// TwinCAT 3 PLC project tmo_motion
// Title: lcls-plc-tmo-motion
// Company: SLAC
// ProjectVersion: 0.0.0
// ProgramVersion: 3.1.4022.7
// CompilerDefines: K
// libraries:
//   LCLS General, * (SLAC)
//   lcls-twincat-motion, * (SLAC)
//   lcls2-cc-lib, * (SLAC)
//   PMPS, * (SLAC - LCLS)
//   Tc2_MC2, * (Beckhoff Automation GmbH)
//   Tc2_SerialCom, * (Beckhoff Automation GmbH)
//   Tc2_Standard, * (Beckhoff Automation GmbH)
//   Tc2_System, * (Beckhoff Automation GmbH)
//   Tc3_Module, * (Beckhoff Automation GmbH)
// project tree:
//   DUTs/ E_HomeState.TcDUT (not stored)
//   GVLs/ GVL_PMPS.TcGVL (not stored), Main.TcGVL
//   / PlcTask.TcTTO
//   POUs/ PRG_1_PlcTask.TcPOU, PRG_2_PMPS_PRE.TcPOU, PRG_3_PMPS_POST.TcPOU, PRG_4_LOG.TcPOU, PRG_AL1K4_L2SI.TcPOU, PRG_IM2K4_PPM.TcPOU, PRG_IM3K4_PPM.TcPOU, PRG_IM4K4_PPM.TcPOU, PRG_IM5K4_PPM.TcPOU, PRG_LI1K4_IP1.TcPOU, PRG_PF1K4_WFS_TARGET.TcPOU, PRG_SL1K4_SCATTER.TcPOU, PRG_SL2K4_SCATTER.TcPOU, PRG_ST4K4_TMO_TERM.TcPOU, PRG_ST5K4_TMO_TERM_FIXED.TcPOU, PRG_TM1K4.TcPOU (not stored)
//   POUs/temp/ FB_SLITS.TcPOU, FB_SLITS_POWER.TcPOU (not stored), FB_SLITS_SCATTER.TcPOU
// real-time tasks:
//   TASK PlcTask: cycle T#10ms, priority 20, ADS port 350
// motion (NC):
//   TASK NC-Task 1 SAF: cycle T#2ms, priority 4, ADS port 501
//   TASK NC-Task 1 SVB: cycle T#10ms, priority 8, ADS port 511
//   AXIS Axis 1 AL1K4-L2SI-MMS (id 1)
//     Dynamic: AccelerationMaximum=200, DecelerationMaximum=200, Acceleration=200, Deceleration=200, Jerk=500, DelayTime=0.004
//     Velo: Maximum=10
//     TargetPosControl: Range=0.002, Time=2
//     OtherSettings: AllowMotionCmdToSlave=true
//     encoder EncType=29
//       EncPara: ScaleFactorNumerator=5e-05, Offset=-214686.941, MaxCount=#xffffffff, ReferenceSystem=1
//         SoftEndMinControl: Enable=true, Range=-108.74
//         SoftEndMaxControl: Enable=true, Range=-33.49
//         Inc: RefSoftSyncMask=#x0000ffff
//     drive DrvType=24
//       Analog: VeloReferenz=100, ScaleFactorActTorque=0.1
//       TimeComp: TaskDelayCycles=1
//     controller CtrType=2
//       CtrPara: PriorControlFactor=1
//         PosDiffControl: Range=1
//         PID: PosKp=20, PosExtKp=1, PosExtVelo=0.1, DeadBandPosition=0.002
//         Observer: BandWidth=20
//   AXIS Axis 2 (id 2)
//     OtherSettings: AllowMotionCmdToSlave=true
//     encoder EncType=1
//     drive DrvType=5
//       Analog: ScaleFactorActTorque=0.1
//       TimeComp: TaskDelayCycles=1
//     controller CtrType=1
//       CtrPara: PriorControlFactor=1
//         Observer: BandWidth=20
//   AXIS Axis 3 (id 3)
//     OtherSettings: AllowMotionCmdToSlave=true
//     encoder EncType=1
//     drive DrvType=5
//       Analog: ScaleFactorActTorque=0.1
//       TimeComp: TaskDelayCycles=1
//     controller CtrType=1
//       CtrPara: PriorControlFactor=1
//         Observer: BandWidth=20
//   AXIS Axis 4 (id 4)
//     OtherSettings: AllowMotionCmdToSlave=true
//     encoder EncType=1
//     drive DrvType=5
//       Analog: ScaleFactorActTorque=0.1
//       TimeComp: TaskDelayCycles=1
//     controller CtrType=1
//       CtrPara: PriorControlFactor=1
//         Observer: BandWidth=20
//   AXIS Axis 5 (id 5)
//     OtherSettings: AllowMotionCmdToSlave=true
//     encoder EncType=1
//     drive DrvType=5
//       Analog: ScaleFactorActTorque=0.1
//       TimeComp: TaskDelayCycles=1
//     controller CtrType=1
//       CtrPara: PriorControlFactor=1
//         Observer: BandWidth=20
//   AXIS Axis 6 IM1K4-XTES-MMS (id 6)
//     Velo: Maximum=10
//     OtherSettings: AllowMotionCmdToSlave=true
//     encoder EncType=29
//       EncPara: ScaleFactorNumerator=5e-05, Offset=-398.1892, MaxCount=#x00400000, ReferenceSystem=1
//         SoftEndMinControl: Enable=true, Range=-90
//         SoftEndMaxControl: Enable=true
//         Inc: RefSoftSyncMask=#x00000000
//     drive DrvType=24
//       DrvPara: Inverse=true
//         Analog: VeloReferenz=50, ScaleFactorActTorque=0.1
//         TimeComp: TaskDelayCycles=1
//     controller CtrType=2
//       CtrPara: PriorControlFactor=1
//         PosDiffControl: Range=1
//         PID: PosKp=20, PosExtKp=20, DeadBandPosition=0.001
//         Observer: BandWidth=20
//   AXIS Axis 7 IM1K4-XTES-CLZ (id 7)
//     General: UnitName=%
//     Velo: Maximum=10
//     OtherSettings: AllowMotionCmdToSlave=true
//     encoder EncType=4
//       EncPara: ScaleFactorNumerator=0.003, MaxCount=#x0000ffff
//         SoftEndMinControl: Enable=true, Range=-100
//         SoftEndMaxControl: Enable=true, Range=100
//         Inc: RefSoftSyncMask=#x0000ffff
//     drive DrvType=23
//       DrvPara: Inverse=true
//         Analog: VeloReferenz=33, ScaleFactorActTorque=0.1
//         TimeComp: TaskDelayCycles=1
//     controller CtrType=2
//       CtrPara: PriorControlFactor=1
//         PosDiffControl: Range=1
//         PID: PosKp=20, PosExtKp=20, DeadBandPosition=0.1
//         Observer: BandWidth=20
//   AXIS Axis 8 IM1K4-XTES-CLF (id 8)
//     General: UnitName=%
//     Velo: Maximum=10
//     OtherSettings: AllowMotionCmdToSlave=true
//     encoder EncType=4
//       EncPara: ScaleFactorNumerator=0.008, MaxCount=#x0000ffff
//         SoftEndMinControl: Enable=true, Range=-100
//         SoftEndMaxControl: Enable=true, Range=100
//         Inc: RefSoftSyncMask=#x0000ffff
//     drive DrvType=23
//       DrvPara: Inverse=true
//         Analog: VeloReferenz=70, ScaleFactorActTorque=0.1
//         TimeComp: TaskDelayCycles=1
//     controller CtrType=2
//       CtrPara: PriorControlFactor=1
//         PosDiffControl: Range=1
//         PID: PosKp=20, PosExtKp=20, DeadBandPosition=0.1
//         Observer: BandWidth=20
//   AXIS Axis 9 IM2K4-PPM-MMS (id 9)
//     Dynamic: AccelerationMaximum=200, DecelerationMaximum=200, Acceleration=200, Deceleration=200, Jerk=500, DelayTime=0.004
//     Velo: Maximum=65
//     TargetPosControl: Range=0.002, Time=2
//     OtherSettings: AllowMotionCmdToSlave=true
//     encoder EncType=29
//       EncPara: ScaleFactorNumerator=5e-05, Offset=-358.0066, MaxCount=#x00400000, ReferenceSystem=1
//         SoftEndMinControl: Enable=true, Range=-100.57
//         SoftEndMaxControl: Enable=true, Range=-7.67
//         Inc: RefSoftSyncMask=#x00000000
//     drive DrvType=24
//       Analog: VeloReferenz=100, ScaleFactorActTorque=0.1
//       TimeComp: TaskDelayCycles=1
//     controller CtrType=2
//       CtrPara: PriorControlFactor=1
//         PosDiffControl: Range=1
//         PID: PosKp=20, PosExtKp=1, PosExtVelo=0.1, DeadBandPosition=0.002
//         Observer: BandWidth=20
//   AXIS SL1K4-BOTTOM-M10 (id 10)
//     Velo: RefSearch=0.2, RefSync=0.05, Maximum=2.2
//     OtherSettings: AllowMotionCmdToSlave=true
//     encoder EncType=4
//       EncPara: MaxCount=#x0000ffff
//         SoftEndMinControl: Enable=true, Range=-31.51
//         SoftEndMaxControl: Enable=true
//         Inc: RefSoftSyncMask=#x0000ffff
//     drive DrvType=24
//       Analog: VeloReferenz=2, ScaleFactorActTorque=0.1
//       TimeComp: TaskDelayCycles=1
//     controller CtrType=1
//       CtrPara: PriorControlFactor=1
//         PosDiffControl: Range=0.05
//         Observer: BandWidth=20
//   AXIS SL1K4-TOP-M11 (id 11)
//     Velo: RefSearch=0.2, RefSync=0.05, Maximum=2.2
//     OtherSettings: AllowMotionCmdToSlave=true
//     encoder EncType=4
//       EncPara: Inverse=true, MaxCount=#x0000ffff
//         SoftEndMinControl: Enable=true, Range=-31.99
//         SoftEndMaxControl: Enable=true
//         Inc: RefSoftSyncMask=#x0000ffff
//     drive DrvType=24
//       Analog: VeloReferenz=2, ScaleFactorActTorque=0.1
//       TimeComp: TaskDelayCycles=1
//     controller CtrType=1
//       CtrPara: PriorControlFactor=1
//         PosDiffControl: Range=0.05
//         Observer: BandWidth=20
//   AXIS SL1K4-NORTH-M12 (id 12)
//     Velo: RefSearch=0.2, RefSync=0.05, Maximum=2.2
//     OtherSettings: AllowMotionCmdToSlave=true
//     encoder EncType=4
//       EncPara: Inverse=true, MaxCount=#x0000ffff
//         SoftEndMinControl: Enable=true, Range=-31.5
//         SoftEndMaxControl: Enable=true
//         Inc: RefSoftSyncMask=#x0000ffff
//     drive DrvType=24
//       Analog: VeloReferenz=2, ScaleFactorActTorque=0.1
//       TimeComp: TaskDelayCycles=1
//     controller CtrType=1
//       CtrPara: PriorControlFactor=1
//         PosDiffControl: Range=0.05
//         Observer: BandWidth=20
//   AXIS SL1K4-SOUTH-M13 (id 13)
//     Velo: RefSearch=0.2, RefSync=0.05, Maximum=2.2
//     OtherSettings: AllowMotionCmdToSlave=true
//     encoder EncType=4
//       EncPara: MaxCount=#x0000ffff
//         SoftEndMinControl: Enable=true, Range=-30.29
//         SoftEndMaxControl: Enable=true
//         Inc: RefSoftSyncMask=#x0000ffff
//     drive DrvType=24
//       Analog: VeloReferenz=2, ScaleFactorActTorque=0.1
//       TimeComp: TaskDelayCycles=1
//     controller CtrType=1
//       CtrPara: PriorControlFactor=1
//         PosDiffControl: Range=0.05
//         Observer: BandWidth=20
//   AXIS ST1K4-TEST (id 14)
//     Velo: RefSearch=5, RefSync=5, SlowManual=1, FastManual=5, Maximum=50
//     OtherSettings: AllowMotionCmdToSlave=true
//     encoder EncType=4
//       EncPara: ScaleFactorNumerator=0.000390625, Inverse=true, MaxCount=#x0000ffff
//         Inc: RefSoftSyncMask=#x0000ffff
//     drive DrvType=24
//       DrvPara: Inverse=true
//         Analog: VeloReferenz=50
//         TimeComp: TaskDelayCycles=1
//     controller CtrType=1
//       CtrPara: PriorControlFactor=1
//         PosDiffControl: Enable=false, Range=0.05
//         Observer: BandWidth=20
//   AXIS Axis 15 IM3K4-PPM-MMS (id 15)
//     Dynamic: AccelerationMaximum=200, DecelerationMaximum=200, Acceleration=200, Deceleration=200, Jerk=500, DelayTime=0.004
//     Velo: Maximum=65
//     TargetPosControl: Range=0.002, Time=2
//     OtherSettings: AllowMotionCmdToSlave=true
//     encoder EncType=29
//       EncPara: ScaleFactorNumerator=5e-05, Offset=-358.0066, MaxCount=#x00400000, ReferenceSystem=1
//         SoftEndMinControl: Enable=true, Range=-97.98
//         SoftEndMaxControl: Enable=true, Range=-5.69
//     drive DrvType=24
//       Analog: VeloReferenz=100, ScaleFactorActTorque=0.1
//       TimeComp: TaskDelayCycles=1
//     controller CtrType=2
//       CtrPara: PriorControlFactor=1
//         PosDiffControl: Range=1
//         PID: PosKp=20, PosExtKp=1, PosExtVelo=0.1, DeadBandPosition=0.002
//         Observer: BandWidth=20
//   AXIS Axis 16 IM4K4-PPM-MMS (id 16)
//     Dynamic: AccelerationMaximum=200, DecelerationMaximum=200, Acceleration=200, Deceleration=200, Jerk=500, DelayTime=0.004
//     Velo: Maximum=65
//     TargetPosControl: Range=0.002, Time=2
//     OtherSettings: AllowMotionCmdToSlave=true
//     encoder EncType=29
//       EncPara: ScaleFactorNumerator=5e-05, Offset=-358.0066, MaxCount=#x00400000, ReferenceSystem=1
//         SoftEndMinControl: Enable=true, Range=-99.53
//         SoftEndMaxControl: Enable=true, Range=-8.43
//     drive DrvType=24
//       Analog: VeloReferenz=100, ScaleFactorActTorque=0.1
//       TimeComp: TaskDelayCycles=1
//     controller CtrType=2
//       CtrPara: PriorControlFactor=1
//         PosDiffControl: Range=1
//         PID: PosKp=20, PosExtKp=1, PosExtVelo=0.1, DeadBandPosition=0.002
//         Observer: BandWidth=20
//   AXIS Axis 17 IM5K4-PPM-MMS (id 17)
//     Dynamic: AccelerationMaximum=200, DecelerationMaximum=200, Acceleration=200, Deceleration=200, Jerk=500, DelayTime=0.004
//     Velo: Maximum=65
//     TargetPosControl: Range=0.002, Time=2
//     OtherSettings: AllowMotionCmdToSlave=true
//     encoder EncType=29
//       EncPara: ScaleFactorNumerator=5e-05, Offset=-358.0066, MaxCount=#x00400000, ReferenceSystem=1
//         SoftEndMinControl: Enable=true, Range=-97.47
//         SoftEndMaxControl: Enable=true, Range=-4.42
//     drive DrvType=24
//       Analog: VeloReferenz=100, ScaleFactorActTorque=0.1
//       TimeComp: TaskDelayCycles=1
//     controller CtrType=2
//       CtrPara: PriorControlFactor=1
//         PosDiffControl: Range=1
//         PID: PosKp=20, PosExtKp=1, PosExtVelo=0.1, DeadBandPosition=0.002
//         Observer: BandWidth=20
//   AXIS Axis 18 PF1K4-WFS_TARGET-MMS-Y (id 18)
//     Dynamic: AccelerationMaximum=200, DecelerationMaximum=200, Acceleration=10, Deceleration=10, Jerk=500, DelayTime=0.004
//     Velo: Maximum=20
//     TargetPosControl: Range=0.002, Time=2
//     OtherSettings: AllowMotionCmdToSlave=true
//     encoder EncType=29
//       EncPara: ScaleFactorNumerator=5e-05, Offset=-358.0066, MaxCount=#x00400000, ReferenceSystem=1
//         SoftEndMinControl: Enable=true, Range=-99.33
//         SoftEndMaxControl: Enable=true, Range=-9.71
//     drive DrvType=24
//       Analog: VeloReferenz=100, ScaleFactorActTorque=0.1
//       TimeComp: TaskDelayCycles=1
//     controller CtrType=2
//       CtrPara: PriorControlFactor=1
//         PosDiffControl: Range=1
//         PID: PosKp=20, PosExtKp=1, PosExtVelo=0.1, DeadBandPosition=0.002
//         Observer: BandWidth=20
//   AXIS Axis 19 PF1K4-WFS_TARGET-MMS-Z (id 19)
//     Dynamic: AccelerationMaximum=200, DecelerationMaximum=200, Acceleration=10, Deceleration=50, Jerk=500
//     Velo: Maximum=5
//     OtherSettings: AllowMotionCmdToSlave=true
//     encoder EncType=29
//       EncPara: ScaleFactorNumerator=5e-05, MaxCount=#x00400000, ReferenceSystem=1
//         SoftEndMinControl: Enable=true, Range=6.5
//         SoftEndMaxControl: Enable=true, Range=56
//     drive DrvType=24
//       DrvPara: Inverse=true
//         Analog: VeloReferenz=15.875, ScaleFactorActTorque=0.1
//         TimeComp: TaskDelayCycles=1
//     controller CtrType=1
//       CtrPara: PriorControlFactor=1
//         PosDiffControl: Range=1
//         Observer: BandWidth=20
//   AXIS Axis 20 LI1K4-IP1-MMS (id 20)
//     Dynamic: AccelerationMaximum=200, DecelerationMaximum=200, Acceleration=200, Deceleration=200, Jerk=500, DelayTime=0.004
//     Velo: Maximum=65
//     TargetPosControl: Range=0.002, Time=2
//     OtherSettings: AllowMotionCmdToSlave=true
//     encoder EncType=29
//       EncPara: ScaleFactorNumerator=5e-05, Offset=-358.0066, MaxCount=#x00400000, ReferenceSystem=1
//         SoftEndMinControl: Enable=true, Range=-107.43
//         SoftEndMaxControl: Enable=true, Range=1.35
//     drive DrvType=24
//       Analog: VeloReferenz=100, ScaleFactorActTorque=0.1
//       TimeComp: TaskDelayCycles=1
//     controller CtrType=2
//       CtrPara: PriorControlFactor=1
//         PosDiffControl: Range=1
//         PID: PosKp=20, PosExtKp=1, PosExtVelo=0.1, DeadBandPosition=0.002
//         Observer: BandWidth=20
//   AXIS Axis 21 TM1K4-MMS-Y (id 21)
//   AXIS Axis 22 TM1K4-MMS-X (id 22)
//   AXIS SL2K4-BOTTOM-M23 (id 23) // C:\Github\lcls-plc-tmo-motion\plc-tmo-motion\_Config\NC\Axes\SL2K4-BOTTOM-M23.xti
//     Velo: RefSearch=0.2, RefSync=0.05, Maximum=2.2
//     OtherSettings: AllowMotionCmdToSlave=true
//     encoder EncType=4
//       EncPara: MaxCount=#x0000ffff
//         SoftEndMinControl: Enable=true, Range=-30.61
//         SoftEndMaxControl: Enable=true
//         Inc: RefSoftSyncMask=#x0000ffff
//     drive DrvType=24
//       Analog: VeloReferenz=2, ScaleFactorActTorque=0.1
//       TimeComp: TaskDelayCycles=1
//     controller CtrType=1
//       CtrPara: PriorControlFactor=1
//         Observer: BandWidth=20
//   AXIS SL2K4-TOP-M24 (id 24) // C:\Github\lcls-plc-tmo-motion\plc-tmo-motion\_Config\NC\Axes\SL2K4-TOP-M24.xti
//     Velo: RefSearch=0.2, RefSync=0.05, Maximum=2.2
//     PositionAreaControl: Range=0.5
//     TargetPosControl: Range=0.1
//     OtherSettings: AllowMotionCmdToSlave=true
//     encoder EncType=4
//       EncPara: Inverse=true, MaxCount=#x0000ffff
//         SoftEndMinControl: Enable=true, Range=-30.91
//         SoftEndMaxControl: Enable=true
//         Inc: RefSoftSyncMask=#x0000ffff
//     drive DrvType=24
//       Analog: VeloReferenz=2, ScaleFactorActTorque=0.1
//       TimeComp: TaskDelayCycles=1
//     controller CtrType=1
//       CtrPara: PriorControlFactor=1
//         PosDiffControl: Range=0.5
//         Observer: BandWidth=20
//   AXIS SL2K4-NORTH-M25 (id 25) // C:\Github\lcls-plc-tmo-motion\plc-tmo-motion\_Config\NC\Axes\SL2K4-NORTH-M25.xti
//     Velo: RefSearch=0.2, RefSync=0.05, Maximum=2.2
//     OtherSettings: AllowMotionCmdToSlave=true
//     encoder EncType=4
//       EncPara: Inverse=true, MaxCount=#x0000ffff
//         SoftEndMinControl: Enable=true, Range=-30.81
//         SoftEndMaxControl: Enable=true
//         Inc: RefSoftSyncMask=#x0000ffff
//     drive DrvType=24
//       Analog: VeloReferenz=2, ScaleFactorActTorque=0.1
//       TimeComp: TaskDelayCycles=1
//     controller CtrType=1
//       CtrPara: PriorControlFactor=1
//         Observer: BandWidth=20
//   AXIS SL2K4-SOUTH-M26 (id 26) // C:\Github\lcls-plc-tmo-motion\plc-tmo-motion\_Config\NC\Axes\SL2K4-SOUTH-M26.xti
//     Velo: RefSearch=0.2, RefSync=0.05, Maximum=2.2
//     OtherSettings: AllowMotionCmdToSlave=true
//     encoder EncType=4
//       EncPara: MaxCount=#x0000ffff
//         SoftEndMinControl: Enable=true, Range=-30.52
//         SoftEndMaxControl: Enable=true
//         Inc: RefSoftSyncMask=#x0000ffff
//     drive DrvType=24
//       Analog: VeloReferenz=2, ScaleFactorActTorque=0.1
//       TimeComp: TaskDelayCycles=1
//     controller CtrType=1
//       CtrPara: PriorControlFactor=1
//         Observer: BandWidth=20
// I/O:
//   DEVICE Device 1 (EtherCAT), AmsNetId 0.0.0.0.2.1
//     Power (EK1200) [EK1200-5000 EtherCAT Power supply (2A E-Bus)]
//       PMPS_FFO
//       License (EL6070)
//       PMPS_PRE [EL6692 EtherCAT Bridge terminal (Primary)]
//       PLC Junction 1 (EK1122) [EK1122 2 port EtherCAT junction]
//         X2 TMO FEE EC2 (EK1100)
//       PLC Junction 2 (EK1122) [EK1122 2 port EtherCAT junction]
//         PLC Coupler 1(EK1100) [EK1100 EtherCAT Coupler (2A E-Bus)]
//           PLC Junction 5 (EK1122)
//           PLC Junction 6 (EK1122)
//         PLC Coupler 2 (EK1100) [EK1100 EtherCAT Coupler (2A E-Bus)]
//           PLC Junction 7 (EK1122)
//           PLC Junction 8 (EK1122)
//           PLC Junction 9 (EK1122)
//           PLC Junction 10 (EK1122)
//       PLC Junction 3 (EK1122)
//       PLC Junction 4 (EK1122)
//       PLC End Coupler (EK1110) [EK1110 EtherCAT extension]
// variable links:
//   Axes/SL1K4-BOTTOM-M10 <-> Device 1 (EtherCAT)/Power (EK1200)/PLC Junction 1 (EK1122)/X2 TMO FEE EC2 (EK1100)/FEE EC2 E1 (EK1122)/X2 SL1K4-SCATTER/SL1K4-EL5101-E2
//     Enc/Inputs/In/nDataIn1[0] <-> ENC Status compact/Counter value
//     Enc/Inputs/In/nDataIn2[0] <-> ENC Status compact/Latch value
//     Enc/Inputs/In/nState1 @bit 4 <-> ENC Status compact/Status/Counter overflow
//     Enc/Inputs/In/nState1 @bit 3 <-> ENC Status compact/Status/Counter underflow
//     Enc/Inputs/In/nState1 @bit 7 <-> ENC Status compact/Status/Extrapolation stall
//     Enc/Inputs/In/nState1 <-> ENC Status compact/Status/Latch C valid
//     Enc/Inputs/In/nState1 @bit 1 <-> ENC Status compact/Status/Latch extern valid
//     Enc/Inputs/In/nState1 @bit 6 <-> ENC Status compact/Status/Open circuit
//     Enc/Inputs/In/nState1 @bit 2 <-> ENC Status compact/Status/Set counter done
//     Enc/Inputs/In/nState1 @bit 5 <-> ENC Status compact/Status/Status of input status
//     Enc/Inputs/In/nState2 @bit 4 <-> ENC Status compact/Status/Status of extern latch
//     Enc/Inputs/In/nState2 <-> ENC Status compact/Status/Status of input A
//     Enc/Inputs/In/nState2 @bit 1 <-> ENC Status compact/Status/Status of input B
//     Enc/Inputs/In/nState2 @bit 2 <-> ENC Status compact/Status/Status of input C
//     Enc/Inputs/In/nState2 @bit 3 <-> ENC Status compact/Status/Status of input gate
//     Enc/Inputs/In/nState2 @bit 5 <-> ENC Status compact/Status/Sync error
//     Enc/Inputs/In/nState2 @bit 6 <-> ENC Status compact/Status/TxPDO State
//     Enc/Inputs/In/nState2 @bit 7 <-> ENC Status compact/Status/TxPDO Toggle
//     Enc/Inputs/In/nState4 @bit 1 <-> WcState/InputToggle
//     Enc/Inputs/In/nState4 <-> WcState/WcState
//     Enc/Outputs/Out/nCtrl1 <-> ENC Control compact/Control/Enable latch C
//     Enc/Outputs/Out/nCtrl1 @bit 3 <-> ENC Control compact/Control/Enable latch extern on negative edge
//     Enc/Outputs/Out/nCtrl1 @bit 1 <-> ENC Control compact/Control/Enable latch extern on positive edge
//     Enc/Outputs/Out/nCtrl1 @bit 2 <-> ENC Control compact/Control/Set counter
//     Enc/Outputs/Out/nDataOut1[0] <-> ENC Control compact/Set counter value
//   Axes/SL1K4-BOTTOM-M10 <-> Device 1 (EtherCAT)/Power (EK1200)/PLC Junction 1 (EK1122)/X2 TMO FEE EC2 (EK1100)/FEE EC2 E1 (EK1122)/X2 SL1K4-SCATTER/SL1K4-EL7031-E1
//     Drive/Inputs/In/nState1 @bit 3 <-> STM Status/Status/Error
//     Drive/Inputs/In/nState1 @bit 5 <-> STM Status/Status/Moving negative
//     Drive/Inputs/In/nState1 @bit 4 <-> STM Status/Status/Moving positive
//     Drive/Inputs/In/nState1 @bit 1 <-> STM Status/Status/Ready
//     Drive/Inputs/In/nState1 <-> STM Status/Status/Ready to enable
//     Drive/Inputs/In/nState1 @bit 6 <-> STM Status/Status/Torque reduced
//     Drive/Inputs/In/nState1 @bit 2 <-> STM Status/Status/Warning
//     Drive/Inputs/In/nState2 @bit 3 <-> STM Status/Status/Digital input 1
//     Drive/Inputs/In/nState2 @bit 4 <-> STM Status/Status/Digital input 2
//     Drive/Inputs/In/nState2 @bit 5 <-> STM Status/Status/Sync error
//     Drive/Inputs/In/nState2 @bit 7 <-> STM Status/Status/TxPDO Toggle
//     Drive/Inputs/In/nState4 @bit 1 <-> WcState/InputToggle
//     Drive/Inputs/In/nState4 <-> WcState/WcState
//     Drive/Outputs/Out/nCtrl1 <-> STM Control/Control/Enable
//     Drive/Outputs/Out/nCtrl1 @bit 2 <-> STM Control/Control/Reduce torque
//     Drive/Outputs/Out/nCtrl1 @bit 1 <-> STM Control/Control/Reset
//     Drive/Outputs/Out/nDataOut2[0] <-> STM Velocity/Velocity
//   Axes/SL1K4-NORTH-M12 <-> Device 1 (EtherCAT)/Power (EK1200)/PLC Junction 1 (EK1122)/X2 TMO FEE EC2 (EK1100)/FEE EC2 E1 (EK1122)/X2 SL1K4-SCATTER/SL1K4-EL5101-E6
//     Enc/Inputs/In/nDataIn1[0] <-> ENC Status compact/Counter value
//     Enc/Inputs/In/nDataIn2[0] <-> ENC Status compact/Latch value
//     Enc/Inputs/In/nState1 @bit 4 <-> ENC Status compact/Status/Counter overflow
//     Enc/Inputs/In/nState1 @bit 3 <-> ENC Status compact/Status/Counter underflow
//     Enc/Inputs/In/nState1 @bit 7 <-> ENC Status compact/Status/Extrapolation stall
//     Enc/Inputs/In/nState1 <-> ENC Status compact/Status/Latch C valid
//     Enc/Inputs/In/nState1 @bit 1 <-> ENC Status compact/Status/Latch extern valid
//     Enc/Inputs/In/nState1 @bit 6 <-> ENC Status compact/Status/Open circuit
//     Enc/Inputs/In/nState1 @bit 2 <-> ENC Status compact/Status/Set counter done
//     Enc/Inputs/In/nState1 @bit 5 <-> ENC Status compact/Status/Status of input status
//     Enc/Inputs/In/nState2 @bit 4 <-> ENC Status compact/Status/Status of extern latch
//     Enc/Inputs/In/nState2 <-> ENC Status compact/Status/Status of input A
//     Enc/Inputs/In/nState2 @bit 1 <-> ENC Status compact/Status/Status of input B
//     Enc/Inputs/In/nState2 @bit 2 <-> ENC Status compact/Status/Status of input C
//     Enc/Inputs/In/nState2 @bit 3 <-> ENC Status compact/Status/Status of input gate
//     Enc/Inputs/In/nState2 @bit 5 <-> ENC Status compact/Status/Sync error
//     Enc/Inputs/In/nState2 @bit 6 <-> ENC Status compact/Status/TxPDO State
//     Enc/Inputs/In/nState2 @bit 7 <-> ENC Status compact/Status/TxPDO Toggle
//     Enc/Inputs/In/nState4 @bit 1 <-> WcState/InputToggle
//     Enc/Inputs/In/nState4 <-> WcState/WcState
//     Enc/Outputs/Out/nCtrl1 <-> ENC Control compact/Control/Enable latch C
//     Enc/Outputs/Out/nCtrl1 @bit 3 <-> ENC Control compact/Control/Enable latch extern on negative edge
//     Enc/Outputs/Out/nCtrl1 @bit 1 <-> ENC Control compact/Control/Enable latch extern on positive edge
//     Enc/Outputs/Out/nCtrl1 @bit 2 <-> ENC Control compact/Control/Set counter
//     Enc/Outputs/Out/nDataOut1[0] <-> ENC Control compact/Set counter value
//   Axes/SL1K4-NORTH-M12 <-> Device 1 (EtherCAT)/Power (EK1200)/PLC Junction 1 (EK1122)/X2 TMO FEE EC2 (EK1100)/FEE EC2 E1 (EK1122)/X2 SL1K4-SCATTER/SL1K4-EL7031-E5
//     Drive/Inputs/In/nState1 @bit 3 <-> STM Status/Status/Error
//     Drive/Inputs/In/nState1 @bit 5 <-> STM Status/Status/Moving negative
//     Drive/Inputs/In/nState1 @bit 4 <-> STM Status/Status/Moving positive
//     Drive/Inputs/In/nState1 @bit 1 <-> STM Status/Status/Ready
//     Drive/Inputs/In/nState1 <-> STM Status/Status/Ready to enable
//     Drive/Inputs/In/nState1 @bit 6 <-> STM Status/Status/Torque reduced
//     Drive/Inputs/In/nState1 @bit 2 <-> STM Status/Status/Warning
//     Drive/Inputs/In/nState2 @bit 3 <-> STM Status/Status/Digital input 1
//     Drive/Inputs/In/nState2 @bit 4 <-> STM Status/Status/Digital input 2
//     Drive/Inputs/In/nState2 @bit 5 <-> STM Status/Status/Sync error
//     Drive/Inputs/In/nState2 @bit 7 <-> STM Status/Status/TxPDO Toggle
//     Drive/Inputs/In/nState4 @bit 1 <-> WcState/InputToggle
//     Drive/Inputs/In/nState4 <-> WcState/WcState
//     Drive/Outputs/Out/nCtrl1 <-> STM Control/Control/Enable
//     Drive/Outputs/Out/nCtrl1 @bit 2 <-> STM Control/Control/Reduce torque
//     Drive/Outputs/Out/nCtrl1 @bit 1 <-> STM Control/Control/Reset
//     Drive/Outputs/Out/nDataOut2[0] <-> STM Velocity/Velocity
//   Axes/SL1K4-SOUTH-M13 <-> Device 1 (EtherCAT)/Power (EK1200)/PLC Junction 1 (EK1122)/X2 TMO FEE EC2 (EK1100)/FEE EC2 E1 (EK1122)/X2 SL1K4-SCATTER/SL1K4-EL5101-E8
//     Enc/Inputs/In/nDataIn1[0] <-> ENC Status compact/Counter value
//     Enc/Inputs/In/nDataIn2[0] <-> ENC Status compact/Latch value
//     Enc/Inputs/In/nState1 @bit 4 <-> ENC Status compact/Status/Counter overflow
//     Enc/Inputs/In/nState1 @bit 3 <-> ENC Status compact/Status/Counter underflow
//     Enc/Inputs/In/nState1 @bit 7 <-> ENC Status compact/Status/Extrapolation stall
//     Enc/Inputs/In/nState1 <-> ENC Status compact/Status/Latch C valid
//     Enc/Inputs/In/nState1 @bit 1 <-> ENC Status compact/Status/Latch extern valid
//     Enc/Inputs/In/nState1 @bit 6 <-> ENC Status compact/Status/Open circuit
//     Enc/Inputs/In/nState1 @bit 2 <-> ENC Status compact/Status/Set counter done
//     Enc/Inputs/In/nState1 @bit 5 <-> ENC Status compact/Status/Status of input status
//     Enc/Inputs/In/nState2 @bit 4 <-> ENC Status compact/Status/Status of extern latch
//     Enc/Inputs/In/nState2 <-> ENC Status compact/Status/Status of input A
//     Enc/Inputs/In/nState2 @bit 1 <-> ENC Status compact/Status/Status of input B
//     Enc/Inputs/In/nState2 @bit 2 <-> ENC Status compact/Status/Status of input C
//     Enc/Inputs/In/nState2 @bit 3 <-> ENC Status compact/Status/Status of input gate
//     Enc/Inputs/In/nState2 @bit 5 <-> ENC Status compact/Status/Sync error
//     Enc/Inputs/In/nState2 @bit 6 <-> ENC Status compact/Status/TxPDO State
//     Enc/Inputs/In/nState2 @bit 7 <-> ENC Status compact/Status/TxPDO Toggle
//     Enc/Inputs/In/nState4 @bit 1 <-> WcState/InputToggle
//     Enc/Inputs/In/nState4 <-> WcState/WcState
//     Enc/Outputs/Out/nCtrl1 <-> ENC Control compact/Control/Enable latch C
//     Enc/Outputs/Out/nCtrl1 @bit 3 <-> ENC Control compact/Control/Enable latch extern on negative edge
//     Enc/Outputs/Out/nCtrl1 @bit 1 <-> ENC Control compact/Control/Enable latch extern on positive edge
//     Enc/Outputs/Out/nCtrl1 @bit 2 <-> ENC Control compact/Control/Set counter
//     Enc/Outputs/Out/nDataOut1[0] <-> ENC Control compact/Set counter value
//   Axes/SL1K4-SOUTH-M13 <-> Device 1 (EtherCAT)/Power (EK1200)/PLC Junction 1 (EK1122)/X2 TMO FEE EC2 (EK1100)/FEE EC2 E1 (EK1122)/X2 SL1K4-SCATTER/SL1K4-EL7031-E7
//     Drive/Inputs/In/nState1 @bit 3 <-> STM Status/Status/Error
//     Drive/Inputs/In/nState1 @bit 5 <-> STM Status/Status/Moving negative
//     Drive/Inputs/In/nState1 @bit 4 <-> STM Status/Status/Moving positive
//     Drive/Inputs/In/nState1 @bit 1 <-> STM Status/Status/Ready
//     Drive/Inputs/In/nState1 <-> STM Status/Status/Ready to enable
//     Drive/Inputs/In/nState1 @bit 6 <-> STM Status/Status/Torque reduced
//     Drive/Inputs/In/nState1 @bit 2 <-> STM Status/Status/Warning
//     Drive/Inputs/In/nState2 @bit 3 <-> STM Status/Status/Digital input 1
//     Drive/Inputs/In/nState2 @bit 4 <-> STM Status/Status/Digital input 2
//     Drive/Inputs/In/nState2 @bit 5 <-> STM Status/Status/Sync error
//     Drive/Inputs/In/nState2 @bit 7 <-> STM Status/Status/TxPDO Toggle
//     Drive/Inputs/In/nState4 @bit 1 <-> WcState/InputToggle
//     Drive/Inputs/In/nState4 <-> WcState/WcState
//     Drive/Outputs/Out/nCtrl1 <-> STM Control/Control/Enable
//     Drive/Outputs/Out/nCtrl1 @bit 2 <-> STM Control/Control/Reduce torque
//     Drive/Outputs/Out/nCtrl1 @bit 1 <-> STM Control/Control/Reset
//     Drive/Outputs/Out/nDataOut2[0] <-> STM Velocity/Velocity
//   Axes/SL1K4-TOP-M11 <-> Device 1 (EtherCAT)/Power (EK1200)/PLC Junction 1 (EK1122)/X2 TMO FEE EC2 (EK1100)/FEE EC2 E1 (EK1122)/X2 SL1K4-SCATTER/SL1K4-EL5101-E4
//     Enc/Inputs/In/nDataIn1[0] <-> ENC Status compact/Counter value
//     Enc/Inputs/In/nDataIn2[0] <-> ENC Status compact/Latch value
//     Enc/Inputs/In/nState1 @bit 4 <-> ENC Status compact/Status/Counter overflow
//     Enc/Inputs/In/nState1 @bit 3 <-> ENC Status compact/Status/Counter underflow
//     Enc/Inputs/In/nState1 @bit 7 <-> ENC Status compact/Status/Extrapolation stall
//     Enc/Inputs/In/nState1 <-> ENC Status compact/Status/Latch C valid
//     Enc/Inputs/In/nState1 @bit 1 <-> ENC Status compact/Status/Latch extern valid
//     Enc/Inputs/In/nState1 @bit 6 <-> ENC Status compact/Status/Open circuit
//     Enc/Inputs/In/nState1 @bit 2 <-> ENC Status compact/Status/Set counter done
//     Enc/Inputs/In/nState1 @bit 5 <-> ENC Status compact/Status/Status of input status
//     Enc/Inputs/In/nState2 @bit 4 <-> ENC Status compact/Status/Status of extern latch
//     Enc/Inputs/In/nState2 <-> ENC Status compact/Status/Status of input A
//     Enc/Inputs/In/nState2 @bit 1 <-> ENC Status compact/Status/Status of input B
//     Enc/Inputs/In/nState2 @bit 2 <-> ENC Status compact/Status/Status of input C
//     Enc/Inputs/In/nState2 @bit 3 <-> ENC Status compact/Status/Status of input gate
//     Enc/Inputs/In/nState2 @bit 5 <-> ENC Status compact/Status/Sync error
//     Enc/Inputs/In/nState2 @bit 6 <-> ENC Status compact/Status/TxPDO State
//     Enc/Inputs/In/nState2 @bit 7 <-> ENC Status compact/Status/TxPDO Toggle
//     Enc/Inputs/In/nState4 @bit 1 <-> WcState/InputToggle
//     Enc/Inputs/In/nState4 <-> WcState/WcState
//     Enc/Outputs/Out/nCtrl1 <-> ENC Control compact/Control/Enable latch C
//     Enc/Outputs/Out/nCtrl1 @bit 3 <-> ENC Control compact/Control/Enable latch extern on negative edge
//     Enc/Outputs/Out/nCtrl1 @bit 1 <-> ENC Control compact/Control/Enable latch extern on positive edge
//     Enc/Outputs/Out/nCtrl1 @bit 2 <-> ENC Control compact/Control/Set counter
//     Enc/Outputs/Out/nDataOut1[0] <-> ENC Control compact/Set counter value
//   Axes/SL1K4-TOP-M11 <-> Device 1 (EtherCAT)/Power (EK1200)/PLC Junction 1 (EK1122)/X2 TMO FEE EC2 (EK1100)/FEE EC2 E1 (EK1122)/X2 SL1K4-SCATTER/SL1K4-EL7031-E3
//     Drive/Inputs/In/nState1 @bit 3 <-> STM Status/Status/Error
//     Drive/Inputs/In/nState1 @bit 5 <-> STM Status/Status/Moving negative
//     Drive/Inputs/In/nState1 @bit 4 <-> STM Status/Status/Moving positive
//     Drive/Inputs/In/nState1 @bit 1 <-> STM Status/Status/Ready
//     Drive/Inputs/In/nState1 <-> STM Status/Status/Ready to enable
//     Drive/Inputs/In/nState1 @bit 6 <-> STM Status/Status/Torque reduced
//     Drive/Inputs/In/nState1 @bit 2 <-> STM Status/Status/Warning
//     Drive/Inputs/In/nState2 @bit 3 <-> STM Status/Status/Digital input 1
//     Drive/Inputs/In/nState2 @bit 4 <-> STM Status/Status/Digital input 2
//     Drive/Inputs/In/nState2 @bit 5 <-> STM Status/Status/Sync error
//     Drive/Inputs/In/nState2 @bit 7 <-> STM Status/Status/TxPDO Toggle
//     Drive/Inputs/In/nState4 @bit 1 <-> WcState/InputToggle
//     Drive/Inputs/In/nState4 <-> WcState/WcState
//     Drive/Outputs/Out/nCtrl1 <-> STM Control/Control/Enable
//     Drive/Outputs/Out/nCtrl1 @bit 2 <-> STM Control/Control/Reduce torque
//     Drive/Outputs/Out/nCtrl1 @bit 1 <-> STM Control/Control/Reset
//     Drive/Outputs/Out/nDataOut2[0] <-> STM Velocity/Velocity
//   (this object) <-> Device 1 (EtherCAT)/Power (EK1200)/PLC Junction 1 (EK1122)/X2 TMO FEE EC2 (EK1100)/FEE EC2 E1 (EK1122)/X1 AL1K4-L2SI (EK1100)/AL1K4-EL5042-E2
//     Enc/Inputs/In/nComState @bit 1 <-> WcState/InputToggle
//     Enc/Inputs/In/nComState <-> WcState/WcState
//     Enc/Inputs/In/nDataIn1 <-> FB Inputs Channel 1/Position
//     Enc/Inputs/In/nState1 @bit 12 <-> FB Inputs Channel 1/Status/Diag
//     Enc/Inputs/In/nState1 @bit 1 <-> FB Inputs Channel 1/Status/Error
//     Enc/Inputs/In/nState1 @bit 14 <-> FB Inputs Channel 1/Status/Input cycle counter
//     Enc/Inputs/In/nState1 @bit 2 <-> FB Inputs Channel 1/Status/Ready
//     Enc/Inputs/In/nState1 @bit 13 <-> FB Inputs Channel 1/Status/TxPDO State
//     Enc/Inputs/In/nState1 <-> FB Inputs Channel 1/Status/Warning
//   (this object) <-> Device 1 (EtherCAT)/Power (EK1200)/PLC Junction 1 (EK1122)/X2 TMO FEE EC2 (EK1100)/FEE EC2 E1 (EK1122)/X1 AL1K4-L2SI (EK1100)/AL1K4-EL7041-E1
//     Drive/Inputs/In/nState1 @bit 3 <-> STM Status/Status/Error
//     Drive/Inputs/In/nState1 @bit 5 <-> STM Status/Status/Moving negative
//     Drive/Inputs/In/nState1 @bit 4 <-> STM Status/Status/Moving positive
//     Drive/Inputs/In/nState1 @bit 1 <-> STM Status/Status/Ready
//     Drive/Inputs/In/nState1 <-> STM Status/Status/Ready to enable
//     Drive/Inputs/In/nState1 @bit 6 <-> STM Status/Status/Torque reduced
//     Drive/Inputs/In/nState1 @bit 2 <-> STM Status/Status/Warning
//     Drive/Inputs/In/nState2 @bit 3 <-> STM Status/Status/Digital input 1
//     Drive/Inputs/In/nState2 @bit 4 <-> STM Status/Status/Digital input 2
//     Drive/Inputs/In/nState2 @bit 5 <-> STM Status/Status/Sync error
//     Drive/Inputs/In/nState2 @bit 7 <-> STM Status/Status/TxPDO Toggle
//     Drive/Inputs/In/nState4 @bit 1 <-> WcState/InputToggle
//     Drive/Inputs/In/nState4 <-> WcState/WcState
//     Drive/Outputs/Out/nCtrl1 <-> STM Control/Control/Enable
//     Drive/Outputs/Out/nCtrl1 @bit 2 <-> STM Control/Control/Reduce torque
//     Drive/Outputs/Out/nCtrl1 @bit 1 <-> STM Control/Control/Reset
//     Drive/Outputs/Out/nDataOut2[0] <-> STM Velocity/Velocity
//   (this object) <-> Device 1 (EtherCAT)/Power (EK1200)/PLC Junction 1 (EK1122)/X2 TMO FEE EC2 (EK1100)/FEE EC2 E2 (EK1122)/X1 IM2K4-PPM (EK1100)/IM2K4-EL5042-E2
//     Enc/Inputs/In/nComState @bit 1 <-> WcState/InputToggle
//     Enc/Inputs/In/nComState <-> WcState/WcState
//     Enc/Inputs/In/nDataIn1 <-> FB Inputs Channel 1/Position
//     Enc/Inputs/In/nState1 @bit 12 <-> FB Inputs Channel 1/Status/Diag
//     Enc/Inputs/In/nState1 @bit 1 <-> FB Inputs Channel 1/Status/Error
//     Enc/Inputs/In/nState1 @bit 14 <-> FB Inputs Channel 1/Status/Input cycle counter
//     Enc/Inputs/In/nState1 @bit 2 <-> FB Inputs Channel 1/Status/Ready
//     Enc/Inputs/In/nState1 @bit 13 <-> FB Inputs Channel 1/Status/TxPDO State
//     Enc/Inputs/In/nState1 <-> FB Inputs Channel 1/Status/Warning
//   (this object) <-> Device 1 (EtherCAT)/Power (EK1200)/PLC Junction 1 (EK1122)/X2 TMO FEE EC2 (EK1100)/FEE EC2 E2 (EK1122)/X1 IM2K4-PPM (EK1100)/IM2K4-EL7041-E1
//     Drive/Inputs/In/nState1 @bit 3 <-> STM Status/Status/Error
//     Drive/Inputs/In/nState1 @bit 5 <-> STM Status/Status/Moving negative
//     Drive/Inputs/In/nState1 @bit 4 <-> STM Status/Status/Moving positive
//     Drive/Inputs/In/nState1 @bit 1 <-> STM Status/Status/Ready
//     Drive/Inputs/In/nState1 <-> STM Status/Status/Ready to enable
//     Drive/Inputs/In/nState1 @bit 6 <-> STM Status/Status/Torque reduced
//     Drive/Inputs/In/nState1 @bit 2 <-> STM Status/Status/Warning
//     Drive/Inputs/In/nState2 @bit 3 <-> STM Status/Status/Digital input 1
//     Drive/Inputs/In/nState2 @bit 4 <-> STM Status/Status/Digital input 2
//     Drive/Inputs/In/nState2 @bit 5 <-> STM Status/Status/Sync error
//     Drive/Inputs/In/nState2 @bit 7 <-> STM Status/Status/TxPDO Toggle
//     Drive/Inputs/In/nState4 @bit 1 <-> WcState/InputToggle
//     Drive/Inputs/In/nState4 <-> WcState/WcState
//     Drive/Outputs/Out/nCtrl1 <-> STM Control/Control/Enable
//     Drive/Outputs/Out/nCtrl1 @bit 2 <-> STM Control/Control/Reduce torque
//     Drive/Outputs/Out/nCtrl1 @bit 1 <-> STM Control/Control/Reset
//     Drive/Outputs/Out/nDataOut2[0] <-> STM Velocity/Velocity
//   (this object) <-> Device 1 (EtherCAT)/Power (EK1200)/PLC Junction 2 (EK1122)/PLC Coupler 1(EK1100)/PLC Junction 5 (EK1122)/IM3K4-PPM (EK1100)/IM3K4-EL5042-E2
//     Enc/Inputs/In/nComState @bit 1 <-> WcState/InputToggle
//     Enc/Inputs/In/nComState <-> WcState/WcState
//     Enc/Inputs/In/nDataIn1 <-> FB Inputs Channel 1/Position
//     Enc/Inputs/In/nState1 @bit 12 <-> FB Inputs Channel 1/Status/Diag
//     Enc/Inputs/In/nState1 @bit 1 <-> FB Inputs Channel 1/Status/Error
//     Enc/Inputs/In/nState1 @bit 14 <-> FB Inputs Channel 1/Status/Input cycle counter
//     Enc/Inputs/In/nState1 @bit 2 <-> FB Inputs Channel 1/Status/Ready
//     Enc/Inputs/In/nState1 @bit 13 <-> FB Inputs Channel 1/Status/TxPDO State
//     Enc/Inputs/In/nState1 <-> FB Inputs Channel 1/Status/Warning
//   (this object) <-> Device 1 (EtherCAT)/Power (EK1200)/PLC Junction 2 (EK1122)/PLC Coupler 1(EK1100)/PLC Junction 5 (EK1122)/IM3K4-PPM (EK1100)/IM3K4-EL7041-E1
//     Drive/Inputs/In/nState1 @bit 3 <-> STM Status/Status/Error
//     Drive/Inputs/In/nState1 @bit 5 <-> STM Status/Status/Moving negative
//     Drive/Inputs/In/nState1 @bit 4 <-> STM Status/Status/Moving positive
//     Drive/Inputs/In/nState1 @bit 1 <-> STM Status/Status/Ready
//     Drive/Inputs/In/nState1 <-> STM Status/Status/Ready to enable
//     Drive/Inputs/In/nState1 @bit 6 <-> STM Status/Status/Torque reduced
//     Drive/Inputs/In/nState1 @bit 2 <-> STM Status/Status/Warning
//     Drive/Inputs/In/nState2 @bit 5 <-> STM Status/Status/Sync error
//     Drive/Inputs/In/nState2 @bit 7 <-> STM Status/Status/TxPDO Toggle
//     Drive/Inputs/In/nState4 @bit 1 <-> WcState/InputToggle
//     Drive/Inputs/In/nState4 <-> WcState/WcState
//     Drive/Outputs/Out/nCtrl1 <-> STM Control/Control/Enable
//     Drive/Outputs/Out/nCtrl1 @bit 2 <-> STM Control/Control/Reduce torque
//     Drive/Outputs/Out/nCtrl1 @bit 1 <-> STM Control/Control/Reset
//     Drive/Outputs/Out/nDataOut2[0] <-> STM Velocity/Velocity
//   (this object) <-> Device 1 (EtherCAT)/Power (EK1200)/PLC Junction 2 (EK1122)/PLC Coupler 1(EK1100)/PLC Junction 5 (EK1122)/IM4K4-PPM (EK1100)/IM4K4-EL5042-E2
//     Enc/Inputs/In/nComState @bit 1 <-> WcState/InputToggle
//     Enc/Inputs/In/nComState <-> WcState/WcState
//     Enc/Inputs/In/nDataIn1 <-> FB Inputs Channel 1/Position
//     Enc/Inputs/In/nState1 @bit 12 <-> FB Inputs Channel 1/Status/Diag
//     Enc/Inputs/In/nState1 @bit 1 <-> FB Inputs Channel 1/Status/Error
//     Enc/Inputs/In/nState1 @bit 14 <-> FB Inputs Channel 1/Status/Input cycle counter
//     Enc/Inputs/In/nState1 @bit 2 <-> FB Inputs Channel 1/Status/Ready
//     Enc/Inputs/In/nState1 @bit 13 <-> FB Inputs Channel 1/Status/TxPDO State
//     Enc/Inputs/In/nState1 <-> FB Inputs Channel 1/Status/Warning
//   (this object) <-> Device 1 (EtherCAT)/Power (EK1200)/PLC Junction 2 (EK1122)/PLC Coupler 1(EK1100)/PLC Junction 5 (EK1122)/IM4K4-PPM (EK1100)/IM4K4-EL7041-E1
//     Drive/Inputs/In/nState1 @bit 3 <-> STM Status/Status/Error
//     Drive/Inputs/In/nState1 @bit 5 <-> STM Status/Status/Moving negative
//     Drive/Inputs/In/nState1 @bit 4 <-> STM Status/Status/Moving positive
//     Drive/Inputs/In/nState1 @bit 1 <-> STM Status/Status/Ready
//     Drive/Inputs/In/nState1 <-> STM Status/Status/Ready to enable
//     Drive/Inputs/In/nState1 @bit 6 <-> STM Status/Status/Torque reduced
//     Drive/Inputs/In/nState1 @bit 2 <-> STM Status/Status/Warning
//     Drive/Inputs/In/nState2 @bit 3 <-> STM Status/Status/Digital input 1
//     Drive/Inputs/In/nState2 @bit 4 <-> STM Status/Status/Digital input 2
//     Drive/Inputs/In/nState2 @bit 5 <-> STM Status/Status/Sync error
//     Drive/Inputs/In/nState2 @bit 7 <-> STM Status/Status/TxPDO Toggle
//     Drive/Inputs/In/nState4 @bit 1 <-> WcState/InputToggle
//     Drive/Inputs/In/nState4 <-> WcState/WcState
//     Drive/Outputs/Out/nCtrl1 <-> STM Control/Control/Enable
//     Drive/Outputs/Out/nCtrl1 @bit 2 <-> STM Control/Control/Reduce torque
//     Drive/Outputs/Out/nCtrl1 @bit 1 <-> STM Control/Control/Reset
//     Drive/Outputs/Out/nDataOut2[0] <-> STM Velocity/Velocity
//   (this object) <-> Device 1 (EtherCAT)/Power (EK1200)/PLC Junction 2 (EK1122)/PLC Coupler 2 (EK1100)/PLC Junction 8 (EK1122)/IM5K4-PPM (EK1100)/IM5K4-EL5042-E2
//     Enc/Inputs/In/nComState @bit 1 <-> WcState/InputToggle
//     Enc/Inputs/In/nComState <-> WcState/WcState
//     Enc/Inputs/In/nDataIn1 <-> FB Inputs Channel 1/Position
//     Enc/Inputs/In/nState1 @bit 12 <-> FB Inputs Channel 1/Status/Diag
//     Enc/Inputs/In/nState1 @bit 1 <-> FB Inputs Channel 1/Status/Error
//     Enc/Inputs/In/nState1 @bit 14 <-> FB Inputs Channel 1/Status/Input cycle counter
//     Enc/Inputs/In/nState1 @bit 2 <-> FB Inputs Channel 1/Status/Ready
//     Enc/Inputs/In/nState1 @bit 13 <-> FB Inputs Channel 1/Status/TxPDO State
//     Enc/Inputs/In/nState1 <-> FB Inputs Channel 1/Status/Warning
//   (this object) <-> Device 1 (EtherCAT)/Power (EK1200)/PLC Junction 2 (EK1122)/PLC Coupler 2 (EK1100)/PLC Junction 8 (EK1122)/IM5K4-PPM (EK1100)/IM5K4-EL7041-E1
//     Drive/Inputs/In/nState1 @bit 3 <-> STM Status/Status/Error
//     Drive/Inputs/In/nState1 @bit 5 <-> STM Status/Status/Moving negative
//     Drive/Inputs/In/nState1 @bit 4 <-> STM Status/Status/Moving positive
//     Drive/Inputs/In/nState1 @bit 1 <-> STM Status/Status/Ready
//     Drive/Inputs/In/nState1 <-> STM Status/Status/Ready to enable
//     Drive/Inputs/In/nState1 @bit 6 <-> STM Status/Status/Torque reduced
//     Drive/Inputs/In/nState1 @bit 2 <-> STM Status/Status/Warning
//     Drive/Inputs/In/nState2 @bit 3 <-> STM Status/Status/Digital input 1
//     Drive/Inputs/In/nState2 @bit 4 <-> STM Status/Status/Digital input 2
//     Drive/Inputs/In/nState2 @bit 5 <-> STM Status/Status/Sync error
//     Drive/Inputs/In/nState2 @bit 7 <-> STM Status/Status/TxPDO Toggle
//     Drive/Inputs/In/nState4 @bit 1 <-> WcState/InputToggle
//     Drive/Inputs/In/nState4 <-> WcState/WcState
//     Drive/Outputs/Out/nCtrl1 <-> STM Control/Control/Enable
//     Drive/Outputs/Out/nCtrl1 @bit 2 <-> STM Control/Control/Reduce torque
//     Drive/Outputs/Out/nCtrl1 @bit 1 <-> STM Control/Control/Reset
//     Drive/Outputs/Out/nDataOut2[0] <-> STM Velocity/Velocity
//   (this object) <-> Device 1 (EtherCAT)/Power (EK1200)/PLC Junction 2 (EK1122)/PLC Coupler 2 (EK1100)/PLC Junction 10 (EK1122)/PF1K4-WFS (EK1100)/PF1K4-EL5042-E3
//     Enc/Inputs/In/nComState @bit 1 <-> WcState/InputToggle
//     Enc/Inputs/In/nComState <-> WcState/WcState
//     Enc/Inputs/In/nDataIn1 <-> FB Inputs Channel 2/Position
//     Enc/Inputs/In/nDataIn1 <-> FB Inputs Channel 1/Position
//     Enc/Inputs/In/nState1 @bit 12 <-> FB Inputs Channel 2/Status/Diag
//     Enc/Inputs/In/nState1 @bit 12 <-> FB Inputs Channel 1/Status/Diag
//     Enc/Inputs/In/nState1 @bit 1 <-> FB Inputs Channel 2/Status/Error
//     Enc/Inputs/In/nState1 @bit 1 <-> FB Inputs Channel 1/Status/Error
//     Enc/Inputs/In/nState1 @bit 14 <-> FB Inputs Channel 2/Status/Input cycle counter
//     Enc/Inputs/In/nState1 @bit 14 <-> FB Inputs Channel 1/Status/Input cycle counter
//     Enc/Inputs/In/nState1 @bit 2 <-> FB Inputs Channel 2/Status/Ready
//     Enc/Inputs/In/nState1 @bit 2 <-> FB Inputs Channel 1/Status/Ready
//     Enc/Inputs/In/nState1 @bit 13 <-> FB Inputs Channel 2/Status/TxPDO State
//     Enc/Inputs/In/nState1 @bit 13 <-> FB Inputs Channel 1/Status/TxPDO State
//     Enc/Inputs/In/nState1 <-> FB Inputs Channel 2/Status/Warning
//     Enc/Inputs/In/nState1 <-> FB Inputs Channel 1/Status/Warning
//   (this object) <-> Device 1 (EtherCAT)/Power (EK1200)/PLC Junction 2 (EK1122)/PLC Coupler 2 (EK1100)/PLC Junction 10 (EK1122)/PF1K4-WFS (EK1100)/PF1K4-EL7041-E1
//     Drive/Inputs/In/nState1 @bit 3 <-> STM Status/Status/Error
//     Drive/Inputs/In/nState1 @bit 5 <-> STM Status/Status/Moving negative
//     Drive/Inputs/In/nState1 @bit 4 <-> STM Status/Status/Moving positive
//     Drive/Inputs/In/nState1 @bit 1 <-> STM Status/Status/Ready
//     Drive/Inputs/In/nState1 <-> STM Status/Status/Ready to enable
//     Drive/Inputs/In/nState1 @bit 6 <-> STM Status/Status/Torque reduced
//     Drive/Inputs/In/nState1 @bit 2 <-> STM Status/Status/Warning
//     Drive/Inputs/In/nState2 @bit 3 <-> STM Status/Status/Digital input 1
//     Drive/Inputs/In/nState2 @bit 4 <-> STM Status/Status/Digital input 2
//     Drive/Inputs/In/nState2 @bit 5 <-> STM Status/Status/Sync error
//     Drive/Inputs/In/nState2 @bit 7 <-> STM Status/Status/TxPDO Toggle
//     Drive/Inputs/In/nState4 @bit 1 <-> WcState/InputToggle
//     Drive/Inputs/In/nState4 <-> WcState/WcState
//     Drive/Outputs/Out/nCtrl1 <-> STM Control/Control/Enable
//     Drive/Outputs/Out/nCtrl1 @bit 2 <-> STM Control/Control/Reduce torque
//     Drive/Outputs/Out/nCtrl1 @bit 1 <-> STM Control/Control/Reset
//     Drive/Outputs/Out/nDataOut2[0] <-> STM Velocity/Velocity
//   (this object) <-> Device 1 (EtherCAT)/Power (EK1200)/PLC Junction 2 (EK1122)/PLC Coupler 2 (EK1100)/PLC Junction 10 (EK1122)/PF1K4-WFS (EK1100)/PF1K4-EL7041-E2
//     Drive/Inputs/In/nState1 @bit 3 <-> STM Status/Status/Error
//     Drive/Inputs/In/nState1 @bit 5 <-> STM Status/Status/Moving negative
//     Drive/Inputs/In/nState1 @bit 4 <-> STM Status/Status/Moving positive
//     Drive/Inputs/In/nState1 @bit 1 <-> STM Status/Status/Ready
//     Drive/Inputs/In/nState1 <-> STM Status/Status/Ready to enable
//     Drive/Inputs/In/nState1 @bit 6 <-> STM Status/Status/Torque reduced
//     Drive/Inputs/In/nState1 @bit 2 <-> STM Status/Status/Warning
//     Drive/Inputs/In/nState2 @bit 3 <-> STM Status/Status/Digital input 1
//     Drive/Inputs/In/nState2 @bit 4 <-> STM Status/Status/Digital input 2
//     Drive/Inputs/In/nState2 @bit 5 <-> STM Status/Status/Sync error
//     Drive/Inputs/In/nState2 @bit 7 <-> STM Status/Status/TxPDO Toggle
//     Drive/Inputs/In/nState4 @bit 1 <-> WcState/InputToggle
//     Drive/Inputs/In/nState4 <-> WcState/WcState
//     Drive/Outputs/Out/nCtrl1 <-> STM Control/Control/Enable
//     Drive/Outputs/Out/nCtrl1 @bit 2 <-> STM Control/Control/Reduce torque
//     Drive/Outputs/Out/nCtrl1 @bit 1 <-> STM Control/Control/Reset
//     Drive/Outputs/Out/nDataOut2[0] <-> STM Velocity/Velocity
//   (this object) <-> Device 1 (EtherCAT)/Power (EK1200)/PLC Junction 2 (EK1122)/PLC Coupler 1(EK1100)/PLC Junction 6 (EK1122)/LI1K4-LIC (EK1100)/LI1K4-EL5042-E2
//     Enc/Inputs/In/nComState @bit 1 <-> WcState/InputToggle
//     Enc/Inputs/In/nComState <-> WcState/WcState
//     Enc/Inputs/In/nDataIn1 <-> FB Inputs Channel 1/Position
//     Enc/Inputs/In/nState1 @bit 12 <-> FB Inputs Channel 1/Status/Diag
//     Enc/Inputs/In/nState1 @bit 1 <-> FB Inputs Channel 1/Status/Error
//     Enc/Inputs/In/nState1 @bit 14 <-> FB Inputs Channel 1/Status/Input cycle counter
//     Enc/Inputs/In/nState1 @bit 2 <-> FB Inputs Channel 1/Status/Ready
//     Enc/Inputs/In/nState1 @bit 13 <-> FB Inputs Channel 1/Status/TxPDO State
//     Enc/Inputs/In/nState1 <-> FB Inputs Channel 1/Status/Warning
//   (this object) <-> Device 1 (EtherCAT)/Power (EK1200)/PLC Junction 2 (EK1122)/PLC Coupler 1(EK1100)/PLC Junction 6 (EK1122)/LI1K4-LIC (EK1100)/LI1K4-EL7041-E1
//     Drive/Inputs/In/nState1 @bit 3 <-> STM Status/Status/Error
//     Drive/Inputs/In/nState1 @bit 5 <-> STM Status/Status/Moving negative
//     Drive/Inputs/In/nState1 @bit 4 <-> STM Status/Status/Moving positive
//     Drive/Inputs/In/nState1 @bit 1 <-> STM Status/Status/Ready
//     Drive/Inputs/In/nState1 <-> STM Status/Status/Ready to enable
//     Drive/Inputs/In/nState1 @bit 6 <-> STM Status/Status/Torque reduced
//     Drive/Inputs/In/nState1 @bit 2 <-> STM Status/Status/Warning
//     Drive/Inputs/In/nState2 @bit 3 <-> STM Status/Status/Digital input 1
//     Drive/Inputs/In/nState2 @bit 4 <-> STM Status/Status/Digital input 2
//     Drive/Inputs/In/nState2 @bit 5 <-> STM Status/Status/Sync error
//     Drive/Inputs/In/nState2 @bit 7 <-> STM Status/Status/TxPDO Toggle
//     Drive/Inputs/In/nState4 @bit 1 <-> WcState/InputToggle
//     Drive/Inputs/In/nState4 <-> WcState/WcState
//     Drive/Outputs/Out/nCtrl1 <-> STM Control/Control/Enable
//     Drive/Outputs/Out/nCtrl1 @bit 2 <-> STM Control/Control/Reduce torque
//     Drive/Outputs/Out/nCtrl1 @bit 1 <-> STM Control/Control/Reset
//     Drive/Outputs/Out/nDataOut2[0] <-> STM Velocity/Velocity
//   (this object) <-> Device 1 (EtherCAT)/Power (EK1200)/PLC Junction 2 (EK1122)/PLC Coupler 2 (EK1100)/PLC Junction 9 (EK1122)/X2 SL2K4-SCATTER/SL2K4-EL5101-E2
//     Enc/Inputs/In/nDataIn1[0] <-> ENC Status compact/Counter value
//     Enc/Inputs/In/nDataIn2[0] <-> ENC Status compact/Latch value
//     Enc/Inputs/In/nState1 @bit 4 <-> ENC Status compact/Status/Counter overflow
//     Enc/Inputs/In/nState1 @bit 3 <-> ENC Status compact/Status/Counter underflow
//     Enc/Inputs/In/nState1 @bit 7 <-> ENC Status compact/Status/Extrapolation stall
//     Enc/Inputs/In/nState1 <-> ENC Status compact/Status/Latch C valid
//     Enc/Inputs/In/nState1 @bit 1 <-> ENC Status compact/Status/Latch extern valid
//     Enc/Inputs/In/nState1 @bit 6 <-> ENC Status compact/Status/Open circuit
//     Enc/Inputs/In/nState1 @bit 2 <-> ENC Status compact/Status/Set counter done
//     Enc/Inputs/In/nState1 @bit 5 <-> ENC Status compact/Status/Status of input status
//     Enc/Inputs/In/nState2 @bit 4 <-> ENC Status compact/Status/Status of extern latch
//     Enc/Inputs/In/nState2 <-> ENC Status compact/Status/Status of input A
//     Enc/Inputs/In/nState2 @bit 1 <-> ENC Status compact/Status/Status of input B
//     Enc/Inputs/In/nState2 @bit 2 <-> ENC Status compact/Status/Status of input C
//     Enc/Inputs/In/nState2 @bit 3 <-> ENC Status compact/Status/Status of input gate
//     Enc/Inputs/In/nState2 @bit 5 <-> ENC Status compact/Status/Sync error
//     Enc/Inputs/In/nState2 @bit 6 <-> ENC Status compact/Status/TxPDO State
//     Enc/Inputs/In/nState2 @bit 7 <-> ENC Status compact/Status/TxPDO Toggle
//     Enc/Inputs/In/nState4 @bit 1 <-> WcState/InputToggle
//     Enc/Inputs/In/nState4 <-> WcState/WcState
//     Enc/Outputs/Out/nCtrl1 <-> ENC Control compact/Control/Enable latch C
//     Enc/Outputs/Out/nCtrl1 @bit 3 <-> ENC Control compact/Control/Enable latch extern on negative edge
//     Enc/Outputs/Out/nCtrl1 @bit 1 <-> ENC Control compact/Control/Enable latch extern on positive edge
//     Enc/Outputs/Out/nCtrl1 @bit 2 <-> ENC Control compact/Control/Set counter
//     Enc/Outputs/Out/nDataOut1[0] <-> ENC Control compact/Set counter value
//   (this object) <-> Device 1 (EtherCAT)/Power (EK1200)/PLC Junction 2 (EK1122)/PLC Coupler 2 (EK1100)/PLC Junction 9 (EK1122)/X2 SL2K4-SCATTER/SL2K4-EL7031-E1
//     Drive/Inputs/In/nState1 @bit 3 <-> STM Status/Status/Error
//     Drive/Inputs/In/nState1 @bit 5 <-> STM Status/Status/Moving negative
//     Drive/Inputs/In/nState1 @bit 4 <-> STM Status/Status/Moving positive
//     Drive/Inputs/In/nState1 @bit 1 <-> STM Status/Status/Ready
//     Drive/Inputs/In/nState1 <-> STM Status/Status/Ready to enable
//     Drive/Inputs/In/nState1 @bit 6 <-> STM Status/Status/Torque reduced
//     Drive/Inputs/In/nState1 @bit 2 <-> STM Status/Status/Warning
//     Drive/Inputs/In/nState2 @bit 3 <-> STM Status/Status/Digital input 1
//     Drive/Inputs/In/nState2 @bit 4 <-> STM Status/Status/Digital input 2
//     Drive/Inputs/In/nState2 @bit 5 <-> STM Status/Status/Sync error
//     Drive/Inputs/In/nState2 @bit 7 <-> STM Status/Status/TxPDO Toggle
//     Drive/Inputs/In/nState4 @bit 1 <-> WcState/InputToggle
//     Drive/Inputs/In/nState4 <-> WcState/WcState
//     Drive/Outputs/Out/nCtrl1 <-> STM Control/Control/Enable
//     Drive/Outputs/Out/nCtrl1 @bit 2 <-> STM Control/Control/Reduce torque
//     Drive/Outputs/Out/nCtrl1 @bit 1 <-> STM Control/Control/Reset
//     Drive/Outputs/Out/nDataOut2[0] <-> STM Velocity/Velocity
//   (this object) <-> Device 1 (EtherCAT)/Power (EK1200)/PLC Junction 2 (EK1122)/PLC Coupler 2 (EK1100)/PLC Junction 9 (EK1122)/X2 SL2K4-SCATTER/SL2K4-EL5101-E4
//     Enc/Inputs/In/nDataIn1[0] <-> ENC Status compact/Counter value
//     Enc/Inputs/In/nDataIn2[0] <-> ENC Status compact/Latch value
//     Enc/Inputs/In/nState1 @bit 4 <-> ENC Status compact/Status/Counter overflow
//     Enc/Inputs/In/nState1 @bit 3 <-> ENC Status compact/Status/Counter underflow
//     Enc/Inputs/In/nState1 @bit 7 <-> ENC Status compact/Status/Extrapolation stall
//     Enc/Inputs/In/nState1 <-> ENC Status compact/Status/Latch C valid
//     Enc/Inputs/In/nState1 @bit 1 <-> ENC Status compact/Status/Latch extern valid
//     Enc/Inputs/In/nState1 @bit 6 <-> ENC Status compact/Status/Open circuit
//     Enc/Inputs/In/nState1 @bit 2 <-> ENC Status compact/Status/Set counter done
//     Enc/Inputs/In/nState1 @bit 5 <-> ENC Status compact/Status/Status of input status
//     Enc/Inputs/In/nState2 @bit 4 <-> ENC Status compact/Status/Status of extern latch
//     Enc/Inputs/In/nState2 <-> ENC Status compact/Status/Status of input A
//     Enc/Inputs/In/nState2 @bit 1 <-> ENC Status compact/Status/Status of input B
//     Enc/Inputs/In/nState2 @bit 2 <-> ENC Status compact/Status/Status of input C
//     Enc/Inputs/In/nState2 @bit 3 <-> ENC Status compact/Status/Status of input gate
//     Enc/Inputs/In/nState2 @bit 5 <-> ENC Status compact/Status/Sync error
//     Enc/Inputs/In/nState2 @bit 6 <-> ENC Status compact/Status/TxPDO State
//     Enc/Inputs/In/nState2 @bit 7 <-> ENC Status compact/Status/TxPDO Toggle
//     Enc/Inputs/In/nState4 @bit 1 <-> WcState/InputToggle
//     Enc/Inputs/In/nState4 <-> WcState/WcState
//     Enc/Outputs/Out/nCtrl1 <-> ENC Control compact/Control/Enable latch C
//     Enc/Outputs/Out/nCtrl1 @bit 3 <-> ENC Control compact/Control/Enable latch extern on negative edge
//     Enc/Outputs/Out/nCtrl1 @bit 1 <-> ENC Control compact/Control/Enable latch extern on positive edge
//     Enc/Outputs/Out/nCtrl1 @bit 2 <-> ENC Control compact/Control/Set counter
//     Enc/Outputs/Out/nDataOut1[0] <-> ENC Control compact/Set counter value
//   (this object) <-> Device 1 (EtherCAT)/Power (EK1200)/PLC Junction 2 (EK1122)/PLC Coupler 2 (EK1100)/PLC Junction 9 (EK1122)/X2 SL2K4-SCATTER/SL2K4-EL7031-E3
//     Drive/Inputs/In/nState1 @bit 3 <-> STM Status/Status/Error
//     Drive/Inputs/In/nState1 @bit 5 <-> STM Status/Status/Moving negative
//     Drive/Inputs/In/nState1 @bit 4 <-> STM Status/Status/Moving positive
//     Drive/Inputs/In/nState1 @bit 1 <-> STM Status/Status/Ready
//     Drive/Inputs/In/nState1 <-> STM Status/Status/Ready to enable
//     Drive/Inputs/In/nState1 @bit 6 <-> STM Status/Status/Torque reduced
//     Drive/Inputs/In/nState1 @bit 2 <-> STM Status/Status/Warning
//     Drive/Inputs/In/nState2 @bit 3 <-> STM Status/Status/Digital input 1
//     Drive/Inputs/In/nState2 @bit 4 <-> STM Status/Status/Digital input 2
//     Drive/Inputs/In/nState2 @bit 5 <-> STM Status/Status/Sync error
//     Drive/Inputs/In/nState2 @bit 7 <-> STM Status/Status/TxPDO Toggle
//     Drive/Inputs/In/nState4 @bit 1 <-> WcState/InputToggle
//     Drive/Inputs/In/nState4 <-> WcState/WcState
//     Drive/Outputs/Out/nCtrl1 <-> STM Control/Control/Enable
//     Drive/Outputs/Out/nCtrl1 @bit 2 <-> STM Control/Control/Reduce torque
//     Drive/Outputs/Out/nCtrl1 @bit 1 <-> STM Control/Control/Reset
//     Drive/Outputs/Out/nDataOut2[0] <-> STM Velocity/Velocity
//   (this object) <-> Device 1 (EtherCAT)/Power (EK1200)/PLC Junction 2 (EK1122)/PLC Coupler 2 (EK1100)/PLC Junction 9 (EK1122)/X2 SL2K4-SCATTER/SL2K4-EL5101-E6
//     Enc/Inputs/In/nDataIn1[0] <-> ENC Status compact/Counter value
//     Enc/Inputs/In/nDataIn2[0] <-> ENC Status compact/Latch value
//     Enc/Inputs/In/nState1 @bit 4 <-> ENC Status compact/Status/Counter overflow
//     Enc/Inputs/In/nState1 @bit 3 <-> ENC Status compact/Status/Counter underflow
//     Enc/Inputs/In/nState1 @bit 7 <-> ENC Status compact/Status/Extrapolation stall
//     Enc/Inputs/In/nState1 <-> ENC Status compact/Status/Latch C valid
//     Enc/Inputs/In/nState1 @bit 1 <-> ENC Status compact/Status/Latch extern valid
//     Enc/Inputs/In/nState1 @bit 6 <-> ENC Status compact/Status/Open circuit
//     Enc/Inputs/In/nState1 @bit 2 <-> ENC Status compact/Status/Set counter done
//     Enc/Inputs/In/nState1 @bit 5 <-> ENC Status compact/Status/Status of input status
//     Enc/Inputs/In/nState2 @bit 4 <-> ENC Status compact/Status/Status of extern latch
//     Enc/Inputs/In/nState2 <-> ENC Status compact/Status/Status of input A
//     Enc/Inputs/In/nState2 @bit 1 <-> ENC Status compact/Status/Status of input B
//     Enc/Inputs/In/nState2 @bit 2 <-> ENC Status compact/Status/Status of input C
//     Enc/Inputs/In/nState2 @bit 3 <-> ENC Status compact/Status/Status of input gate
//     Enc/Inputs/In/nState2 @bit 5 <-> ENC Status compact/Status/Sync error
//     Enc/Inputs/In/nState2 @bit 6 <-> ENC Status compact/Status/TxPDO State
//     Enc/Inputs/In/nState2 @bit 7 <-> ENC Status compact/Status/TxPDO Toggle
//     Enc/Inputs/In/nState4 @bit 1 <-> WcState/InputToggle
//     Enc/Inputs/In/nState4 <-> WcState/WcState
//     Enc/Outputs/Out/nCtrl1 <-> ENC Control compact/Control/Enable latch C
//     Enc/Outputs/Out/nCtrl1 @bit 3 <-> ENC Control compact/Control/Enable latch extern on negative edge
//     Enc/Outputs/Out/nCtrl1 @bit 1 <-> ENC Control compact/Control/Enable latch extern on positive edge
//     Enc/Outputs/Out/nCtrl1 @bit 2 <-> ENC Control compact/Control/Set counter
//     Enc/Outputs/Out/nDataOut1[0] <-> ENC Control compact/Set counter value
//   (this object) <-> Device 1 (EtherCAT)/Power (EK1200)/PLC Junction 2 (EK1122)/PLC Coupler 2 (EK1100)/PLC Junction 9 (EK1122)/X2 SL2K4-SCATTER/SL2K4-EL7031-E5
//     Drive/Inputs/In/nState1 @bit 3 <-> STM Status/Status/Error
//     Drive/Inputs/In/nState1 @bit 5 <-> STM Status/Status/Moving negative
//     Drive/Inputs/In/nState1 @bit 4 <-> STM Status/Status/Moving positive
//     Drive/Inputs/In/nState1 @bit 1 <-> STM Status/Status/Ready
//     Drive/Inputs/In/nState1 <-> STM Status/Status/Ready to enable
//     Drive/Inputs/In/nState1 @bit 6 <-> STM Status/Status/Torque reduced
//     Drive/Inputs/In/nState1 @bit 2 <-> STM Status/Status/Warning
//     Drive/Inputs/In/nState2 @bit 3 <-> STM Status/Status/Digital input 1
//     Drive/Inputs/In/nState2 @bit 4 <-> STM Status/Status/Digital input 2
//     Drive/Inputs/In/nState2 @bit 5 <-> STM Status/Status/Sync error
//     Drive/Inputs/In/nState2 @bit 7 <-> STM Status/Status/TxPDO Toggle
//     Drive/Inputs/In/nState4 @bit 1 <-> WcState/InputToggle
//     Drive/Inputs/In/nState4 <-> WcState/WcState
//     Drive/Outputs/Out/nCtrl1 <-> STM Control/Control/Enable
//     Drive/Outputs/Out/nCtrl1 @bit 2 <-> STM Control/Control/Reduce torque
//     Drive/Outputs/Out/nCtrl1 @bit 1 <-> STM Control/Control/Reset
//     Drive/Outputs/Out/nDataOut2[0] <-> STM Velocity/Velocity
//   (this object) <-> Device 1 (EtherCAT)/Power (EK1200)/PLC Junction 2 (EK1122)/PLC Coupler 2 (EK1100)/PLC Junction 9 (EK1122)/X2 SL2K4-SCATTER/SL2K4-EL5101-E8
//     Enc/Inputs/In/nDataIn1[0] <-> ENC Status compact/Counter value
//     Enc/Inputs/In/nDataIn2[0] <-> ENC Status compact/Latch value
//     Enc/Inputs/In/nState1 @bit 4 <-> ENC Status compact/Status/Counter overflow
//     Enc/Inputs/In/nState1 @bit 3 <-> ENC Status compact/Status/Counter underflow
//     Enc/Inputs/In/nState1 @bit 7 <-> ENC Status compact/Status/Extrapolation stall
//     Enc/Inputs/In/nState1 <-> ENC Status compact/Status/Latch C valid
//     Enc/Inputs/In/nState1 @bit 1 <-> ENC Status compact/Status/Latch extern valid
//     Enc/Inputs/In/nState1 @bit 6 <-> ENC Status compact/Status/Open circuit
//     Enc/Inputs/In/nState1 @bit 2 <-> ENC Status compact/Status/Set counter done
//     Enc/Inputs/In/nState1 @bit 5 <-> ENC Status compact/Status/Status of input status
//     Enc/Inputs/In/nState2 @bit 4 <-> ENC Status compact/Status/Status of extern latch
//     Enc/Inputs/In/nState2 <-> ENC Status compact/Status/Status of input A
//     Enc/Inputs/In/nState2 @bit 1 <-> ENC Status compact/Status/Status of input B
//     Enc/Inputs/In/nState2 @bit 2 <-> ENC Status compact/Status/Status of input C
//     Enc/Inputs/In/nState2 @bit 3 <-> ENC Status compact/Status/Status of input gate
//     Enc/Inputs/In/nState2 @bit 5 <-> ENC Status compact/Status/Sync error
//     Enc/Inputs/In/nState2 @bit 6 <-> ENC Status compact/Status/TxPDO State
//     Enc/Inputs/In/nState2 @bit 7 <-> ENC Status compact/Status/TxPDO Toggle
//     Enc/Inputs/In/nState4 @bit 1 <-> WcState/InputToggle
//     Enc/Inputs/In/nState4 <-> WcState/WcState
//     Enc/Outputs/Out/nCtrl1 <-> ENC Control compact/Control/Enable latch C
//     Enc/Outputs/Out/nCtrl1 @bit 3 <-> ENC Control compact/Control/Enable latch extern on negative edge
//     Enc/Outputs/Out/nCtrl1 @bit 1 <-> ENC Control compact/Control/Enable latch extern on positive edge
//     Enc/Outputs/Out/nCtrl1 @bit 2 <-> ENC Control compact/Control/Set counter
//     Enc/Outputs/Out/nDataOut1[0] <-> ENC Control compact/Set counter value
//   (this object) <-> Device 1 (EtherCAT)/Power (EK1200)/PLC Junction 2 (EK1122)/PLC Coupler 2 (EK1100)/PLC Junction 9 (EK1122)/X2 SL2K4-SCATTER/SL2K4-EL7031-E7
//     Drive/Inputs/In/nState1 @bit 3 <-> STM Status/Status/Error
//     Drive/Inputs/In/nState1 @bit 5 <-> STM Status/Status/Moving negative
//     Drive/Inputs/In/nState1 @bit 4 <-> STM Status/Status/Moving positive
//     Drive/Inputs/In/nState1 @bit 1 <-> STM Status/Status/Ready
//     Drive/Inputs/In/nState1 <-> STM Status/Status/Ready to enable
//     Drive/Inputs/In/nState1 @bit 6 <-> STM Status/Status/Torque reduced
//     Drive/Inputs/In/nState1 @bit 2 <-> STM Status/Status/Warning
//     Drive/Inputs/In/nState2 @bit 3 <-> STM Status/Status/Digital input 1
//     Drive/Inputs/In/nState2 @bit 4 <-> STM Status/Status/Digital input 2
//     Drive/Inputs/In/nState2 @bit 5 <-> STM Status/Status/Sync error
//     Drive/Inputs/In/nState2 @bit 7 <-> STM Status/Status/TxPDO Toggle
//     Drive/Inputs/In/nState4 @bit 1 <-> WcState/InputToggle
//     Drive/Inputs/In/nState4 <-> WcState/WcState
//     Drive/Outputs/Out/nCtrl1 <-> STM Control/Control/Enable
//     Drive/Outputs/Out/nCtrl1 @bit 2 <-> STM Control/Control/Reduce torque
//     Drive/Outputs/Out/nCtrl1 @bit 1 <-> STM Control/Control/Reset
//     Drive/Outputs/Out/nDataOut2[0] <-> STM Velocity/Velocity
//   tmo_motion Instance <-> Device 1 (EtherCAT)/Power (EK1200)/PLC Junction 1 (EK1122)/X2 TMO FEE EC2 (EK1100)/FEE EC2 E1 (EK1122)/X1 AL1K4-L2SI (EK1100)/AL1K4-EL2004-E3
//     PlcTask Outputs/Main.M1.bBrakeRelease <-> Channel 1/Output
//   tmo_motion Instance <-> Device 1 (EtherCAT)/Power (EK1200)/PLC Junction 1 (EK1122)/X2 TMO FEE EC2 (EK1100)/FEE EC2 E1 (EK1122)/X1 AL1K4-L2SI (EK1100)/AL1K4-EL4004-E4
//     PlcTask Outputs/PRG_AL1K4_L2SI.fbAL1K4.fbLaser.iLaserINT <-> AO Outputs Channel 1/Analog output
//     PlcTask Outputs/PRG_AL1K4_L2SI.fbAL1K4.fbLaser.iShutdownINT <-> AO Outputs Channel 2/Analog output
//   tmo_motion Instance <-> Device 1 (EtherCAT)/Power (EK1200)/PLC Junction 1 (EK1122)/X2 TMO FEE EC2 (EK1100)/FEE EC2 E1 (EK1122)/X1 AL1K4-L2SI (EK1100)/AL1K4-EL5042-E2
//     PlcTask Inputs/Main.M1.nRawEncoderULINT <-> FB Inputs Channel 1/Position
//   tmo_motion Instance <-> Device 1 (EtherCAT)/Power (EK1200)/PLC Junction 1 (EK1122)/X2 TMO FEE EC2 (EK1100)/FEE EC2 E1 (EK1122)/X1 AL1K4-L2SI (EK1100)/AL1K4-EL7041-E1
//     PlcTask Inputs/Main.M1.bLimitBackwardEnable <-> STM Status/Status/Digital input 2
//     PlcTask Inputs/Main.M1.bLimitForwardEnable <-> STM Status/Status/Digital input 1
//   tmo_motion Instance <-> Device 1 (EtherCAT)/Power (EK1200)/PLC Junction 1 (EK1122)/X2 TMO FEE EC2 (EK1100)/FEE EC2 E1 (EK1122)/X2 SL1K4-SCATTER/SL1K4-EL5101-E2
//     PlcTask Inputs/Main.M10.nRawEncoderUINT <-> ENC Status compact/Counter value
//   tmo_motion Instance <-> Device 1 (EtherCAT)/Power (EK1200)/PLC Junction 1 (EK1122)/X2 TMO FEE EC2 (EK1100)/FEE EC2 E1 (EK1122)/X2 SL1K4-SCATTER/SL1K4-EL5101-E4
//     PlcTask Inputs/Main.M11.nRawEncoderUINT <-> ENC Status compact/Counter value
//   tmo_motion Instance <-> Device 1 (EtherCAT)/Power (EK1200)/PLC Junction 1 (EK1122)/X2 TMO FEE EC2 (EK1100)/FEE EC2 E1 (EK1122)/X2 SL1K4-SCATTER/SL1K4-EL5101-E6
//     PlcTask Inputs/Main.M12.nRawEncoderUINT <-> ENC Status compact/Counter value
//   tmo_motion Instance <-> Device 1 (EtherCAT)/Power (EK1200)/PLC Junction 1 (EK1122)/X2 TMO FEE EC2 (EK1100)/FEE EC2 E1 (EK1122)/X2 SL1K4-SCATTER/SL1K4-EL5101-E8
//     PlcTask Inputs/Main.M13.nRawEncoderUINT <-> ENC Status compact/Counter value
//   tmo_motion Instance <-> Device 1 (EtherCAT)/Power (EK1200)/PLC Junction 1 (EK1122)/X2 TMO FEE EC2 (EK1100)/FEE EC2 E1 (EK1122)/X2 SL1K4-SCATTER/SL1K4-EL7031-E1
//     PlcTask Inputs/Main.M10.bLimitBackwardEnable <-> STM Status/Status/Digital input 1
//     PlcTask Inputs/Main.M10.bLimitForwardEnable <-> STM Status/Status/Digital input 2
//   tmo_motion Instance <-> Device 1 (EtherCAT)/Power (EK1200)/PLC Junction 1 (EK1122)/X2 TMO FEE EC2 (EK1100)/FEE EC2 E1 (EK1122)/X2 SL1K4-SCATTER/SL1K4-EL7031-E3
//     PlcTask Inputs/Main.M11.bLimitBackwardEnable <-> STM Status/Status/Digital input 1
//     PlcTask Inputs/Main.M11.bLimitForwardEnable <-> STM Status/Status/Digital input 2
//   tmo_motion Instance <-> Device 1 (EtherCAT)/Power (EK1200)/PLC Junction 1 (EK1122)/X2 TMO FEE EC2 (EK1100)/FEE EC2 E1 (EK1122)/X2 SL1K4-SCATTER/SL1K4-EL7031-E5
//     PlcTask Inputs/Main.M12.bLimitBackwardEnable <-> STM Status/Status/Digital input 2
//     PlcTask Inputs/Main.M12.bLimitForwardEnable <-> STM Status/Status/Digital input 1
//   tmo_motion Instance <-> Device 1 (EtherCAT)/Power (EK1200)/PLC Junction 1 (EK1122)/X2 TMO FEE EC2 (EK1100)/FEE EC2 E1 (EK1122)/X2 SL1K4-SCATTER/SL1K4-EL7031-E7
//     PlcTask Inputs/Main.M13.bLimitBackwardEnable <-> STM Status/Status/Digital input 2
//     PlcTask Inputs/Main.M13.bLimitForwardEnable <-> STM Status/Status/Digital input 1
//   tmo_motion Instance <-> Device 1 (EtherCAT)/Power (EK1200)/PLC Junction 1 (EK1122)/X2 TMO FEE EC2 (EK1100)/FEE EC2 E2 (EK1122)/X1 IM2K4-PPM (EK1100)/IM2K4-EL2004-E3
//     PlcTask Outputs/Main.M9.bBrakeRelease <-> Channel 1/Output
//     PlcTask Outputs/PRG_IM2K4_PPM.fbIM2K4.fbGige.bGigePower <-> Channel 2/Output
//   tmo_motion Instance <-> Device 1 (EtherCAT)/Power (EK1200)/PLC Junction 1 (EK1122)/X2 TMO FEE EC2 (EK1100)/FEE EC2 E2 (EK1122)/X1 IM2K4-PPM (EK1100)/IM2K4-EL3062-E6
//     PlcTask Inputs/PRG_IM2K4_PPM.fbIM2K4.fbPowerMeter.iVoltageINT <-> AI Standard Channel 1/Value
//   tmo_motion Instance <-> Device 1 (EtherCAT)/Power (EK1200)/PLC Junction 1 (EK1122)/X2 TMO FEE EC2 (EK1100)/FEE EC2 E2 (EK1122)/X1 IM2K4-PPM (EK1100)/IM2K4-EL3314-E4
//     PlcTask Inputs/PRG_IM2K4_PPM.fbIM2K4.fbPowerMeter.fbThermoCouple.bError <-> TC Inputs Channel 1/Status/Error
//     PlcTask Inputs/PRG_IM2K4_PPM.fbIM2K4.fbPowerMeter.fbThermoCouple.bOverrange <-> TC Inputs Channel 1/Status/Overrange
//     PlcTask Inputs/PRG_IM2K4_PPM.fbIM2K4.fbPowerMeter.fbThermoCouple.bUnderrange <-> TC Inputs Channel 1/Status/Underrange
//     PlcTask Inputs/PRG_IM2K4_PPM.fbIM2K4.fbPowerMeter.fbThermoCouple.iRaw <-> TC Inputs Channel 1/Value
//     PlcTask Inputs/PRG_IM2K4_PPM.fbIM2K4.fbYagThermoCouple.bError <-> TC Inputs Channel 2/Status/Error
//     PlcTask Inputs/PRG_IM2K4_PPM.fbIM2K4.fbYagThermoCouple.bOverrange <-> TC Inputs Channel 2/Status/Overrange
//     PlcTask Inputs/PRG_IM2K4_PPM.fbIM2K4.fbYagThermoCouple.bUnderrange <-> TC Inputs Channel 2/Status/Underrange
//     PlcTask Inputs/PRG_IM2K4_PPM.fbIM2K4.fbYagThermoCouple.iRaw <-> TC Inputs Channel 2/Value
//   tmo_motion Instance <-> Device 1 (EtherCAT)/Power (EK1200)/PLC Junction 1 (EK1122)/X2 TMO FEE EC2 (EK1100)/FEE EC2 E2 (EK1122)/X1 IM2K4-PPM (EK1100)/IM2K4-EL4004-E7
//     PlcTask Outputs/PRG_IM2K4_PPM.fbIM2K4.fbGige.iIlluminatorINT <-> AO Outputs Channel 1/Analog output
//   tmo_motion Instance <-> Device 1 (EtherCAT)/Power (EK1200)/PLC Junction 1 (EK1122)/X2 TMO FEE EC2 (EK1100)/FEE EC2 E2 (EK1122)/X1 IM2K4-PPM (EK1100)/IM2K4-EL5042-E2
//     PlcTask Inputs/Main.M9.nRawEncoderULINT <-> FB Inputs Channel 1/Position
//   tmo_motion Instance <-> Device 1 (EtherCAT)/Power (EK1200)/PLC Junction 1 (EK1122)/X2 TMO FEE EC2 (EK1100)/FEE EC2 E2 (EK1122)/X1 IM2K4-PPM (EK1100)/IM2K4-EL7041-E1
//     PlcTask Inputs/Main.M9.bLimitBackwardEnable <-> STM Status/Status/Digital input 2
//     PlcTask Inputs/Main.M9.bLimitForwardEnable <-> STM Status/Status/Digital input 1
//   tmo_motion Instance <-> Device 1 (EtherCAT)/Power (EK1200)/PLC Junction 2 (EK1122)/PLC Coupler 1(EK1100)/PLC Junction 5 (EK1122)/IM3K4-PPM (EK1100)/IM3K4-EL2004-E3
//     PlcTask Outputs/Main.M15.bBrakeRelease <-> Channel 1/Output
//     PlcTask Outputs/PRG_IM3K4_PPM.fbIM3K4.fbGige.bGigePower <-> Channel 2/Output
//   tmo_motion Instance <-> Device 1 (EtherCAT)/Power (EK1200)/PLC Junction 2 (EK1122)/PLC Coupler 1(EK1100)/PLC Junction 5 (EK1122)/IM3K4-PPM (EK1100)/IM3K4-EL3062-E6
//     PlcTask Inputs/PRG_IM3K4_PPM.fbIM3K4.fbPowerMeter.iVoltageINT <-> AI Standard Channel 1/Value
//   tmo_motion Instance <-> Device 1 (EtherCAT)/Power (EK1200)/PLC Junction 2 (EK1122)/PLC Coupler 1(EK1100)/PLC Junction 5 (EK1122)/IM3K4-PPM (EK1100)/IM3K4-EL3314-E4
//     PlcTask Inputs/PRG_IM3K4_PPM.fbIM3K4.fbPowerMeter.fbThermoCouple.bError <-> TC Inputs Channel 1/Status/Error
//     PlcTask Inputs/PRG_IM3K4_PPM.fbIM3K4.fbPowerMeter.fbThermoCouple.bOverrange <-> TC Inputs Channel 1/Status/Overrange
//     PlcTask Inputs/PRG_IM3K4_PPM.fbIM3K4.fbPowerMeter.fbThermoCouple.bUnderrange <-> TC Inputs Channel 1/Status/Underrange
//     PlcTask Inputs/PRG_IM3K4_PPM.fbIM3K4.fbPowerMeter.fbThermoCouple.iRaw <-> TC Inputs Channel 1/Value
//     PlcTask Inputs/PRG_IM3K4_PPM.fbIM3K4.fbYagThermoCouple.bError <-> TC Inputs Channel 2/Status/Error
//     PlcTask Inputs/PRG_IM3K4_PPM.fbIM3K4.fbYagThermoCouple.bOverrange <-> TC Inputs Channel 2/Status/Overrange
//     PlcTask Inputs/PRG_IM3K4_PPM.fbIM3K4.fbYagThermoCouple.bUnderrange <-> TC Inputs Channel 2/Status/Underrange
//     PlcTask Inputs/PRG_IM3K4_PPM.fbIM3K4.fbYagThermoCouple.iRaw <-> TC Inputs Channel 2/Value
//   tmo_motion Instance <-> Device 1 (EtherCAT)/Power (EK1200)/PLC Junction 2 (EK1122)/PLC Coupler 1(EK1100)/PLC Junction 5 (EK1122)/IM3K4-PPM (EK1100)/IM3K4-EL4004-E7
//     PlcTask Outputs/PRG_IM3K4_PPM.fbIM3K4.fbGige.iIlluminatorINT <-> AO Outputs Channel 1/Analog output
//   tmo_motion Instance <-> Device 1 (EtherCAT)/Power (EK1200)/PLC Junction 2 (EK1122)/PLC Coupler 1(EK1100)/PLC Junction 5 (EK1122)/IM3K4-PPM (EK1100)/IM3K4-EL5042-E2
//     PlcTask Inputs/Main.M15.nRawEncoderULINT <-> FB Inputs Channel 1/Position
//   tmo_motion Instance <-> Device 1 (EtherCAT)/Power (EK1200)/PLC Junction 2 (EK1122)/PLC Coupler 1(EK1100)/PLC Junction 5 (EK1122)/IM3K4-PPM (EK1100)/IM3K4-EL7041-E1
//     PlcTask Inputs/Main.M15.bLimitBackwardEnable <-> STM Status/Status/Digital input 2
//     PlcTask Inputs/Main.M15.bLimitForwardEnable <-> STM Status/Status/Digital input 1
//   tmo_motion Instance <-> Device 1 (EtherCAT)/Power (EK1200)/PLC Junction 2 (EK1122)/PLC Coupler 1(EK1100)/PLC Junction 5 (EK1122)/IM4K4-PPM (EK1100)/IM4K4-EL2004-E3
//     PlcTask Outputs/Main.M16.bBrakeRelease <-> Channel 1/Output
//     PlcTask Outputs/PRG_IM4K4_PPM.fbIM4K4.fbGige.bGigePower <-> Channel 2/Output
//   tmo_motion Instance <-> Device 1 (EtherCAT)/Power (EK1200)/PLC Junction 2 (EK1122)/PLC Coupler 1(EK1100)/PLC Junction 5 (EK1122)/IM4K4-PPM (EK1100)/IM4K4-EL3062-E6
//     PlcTask Inputs/PRG_IM4K4_PPM.fbIM4K4.fbPowerMeter.iVoltageINT <-> AI Standard Channel 1/Value
//   tmo_motion Instance <-> Device 1 (EtherCAT)/Power (EK1200)/PLC Junction 2 (EK1122)/PLC Coupler 1(EK1100)/PLC Junction 5 (EK1122)/IM4K4-PPM (EK1100)/IM4K4-EL3314-E4
//     PlcTask Inputs/PRG_IM4K4_PPM.fbIM4K4.fbPowerMeter.fbThermoCouple.bError <-> TC Inputs Channel 1/Status/Error
//     PlcTask Inputs/PRG_IM4K4_PPM.fbIM4K4.fbPowerMeter.fbThermoCouple.bOverrange <-> TC Inputs Channel 1/Status/Overrange
//     PlcTask Inputs/PRG_IM4K4_PPM.fbIM4K4.fbPowerMeter.fbThermoCouple.bUnderrange <-> TC Inputs Channel 1/Status/Underrange
//     PlcTask Inputs/PRG_IM4K4_PPM.fbIM4K4.fbPowerMeter.fbThermoCouple.iRaw <-> TC Inputs Channel 1/Value
//     PlcTask Inputs/PRG_IM4K4_PPM.fbIM4K4.fbYagThermoCouple.bError <-> TC Inputs Channel 2/Status/Error
//     PlcTask Inputs/PRG_IM4K4_PPM.fbIM4K4.fbYagThermoCouple.bOverrange <-> TC Inputs Channel 2/Status/Overrange
//     PlcTask Inputs/PRG_IM4K4_PPM.fbIM4K4.fbYagThermoCouple.bUnderrange <-> TC Inputs Channel 2/Status/Underrange
//     PlcTask Inputs/PRG_IM4K4_PPM.fbIM4K4.fbYagThermoCouple.iRaw <-> TC Inputs Channel 2/Value
//   tmo_motion Instance <-> Device 1 (EtherCAT)/Power (EK1200)/PLC Junction 2 (EK1122)/PLC Coupler 1(EK1100)/PLC Junction 5 (EK1122)/IM4K4-PPM (EK1100)/IM4K4-EL4004-E7
//     PlcTask Outputs/PRG_IM4K4_PPM.fbIM4K4.fbGige.iIlluminatorINT <-> AO Outputs Channel 1/Analog output
//   tmo_motion Instance <-> Device 1 (EtherCAT)/Power (EK1200)/PLC Junction 2 (EK1122)/PLC Coupler 1(EK1100)/PLC Junction 5 (EK1122)/IM4K4-PPM (EK1100)/IM4K4-EL5042-E2
//     PlcTask Inputs/Main.M16.nRawEncoderULINT <-> FB Inputs Channel 1/Position
//   tmo_motion Instance <-> Device 1 (EtherCAT)/Power (EK1200)/PLC Junction 2 (EK1122)/PLC Coupler 1(EK1100)/PLC Junction 5 (EK1122)/IM4K4-PPM (EK1100)/IM4K4-EL7041-E1
//     PlcTask Inputs/Main.M16.bLimitBackwardEnable <-> STM Status/Status/Digital input 2
//     PlcTask Inputs/Main.M16.bLimitForwardEnable <-> STM Status/Status/Digital input 1
//   tmo_motion Instance <-> Device 1 (EtherCAT)/Power (EK1200)/PLC Junction 2 (EK1122)/PLC Coupler 1(EK1100)/PLC Junction 6 (EK1122)/LI1K4-LIC (EK1100)/LI1K4-EL2004-E3
//     PlcTask Outputs/Main.M20.bBrakeRelease <-> Channel 1/Output
//   tmo_motion Instance <-> Device 1 (EtherCAT)/Power (EK1200)/PLC Junction 2 (EK1122)/PLC Coupler 1(EK1100)/PLC Junction 6 (EK1122)/LI1K4-LIC (EK1100)/LI1K4-EL5042-E2
//     PlcTask Inputs/Main.M20.nRawEncoderULINT <-> FB Inputs Channel 1/Position
//   tmo_motion Instance <-> Device 1 (EtherCAT)/Power (EK1200)/PLC Junction 2 (EK1122)/PLC Coupler 1(EK1100)/PLC Junction 6 (EK1122)/LI1K4-LIC (EK1100)/LI1K4-EL7041-E1
//     PlcTask Inputs/Main.M20.bLimitBackwardEnable <-> STM Status/Status/Digital input 2
//     PlcTask Inputs/Main.M20.bLimitForwardEnable <-> STM Status/Status/Digital input 1
//   tmo_motion Instance <-> Device 1 (EtherCAT)/Power (EK1200)/PLC Junction 2 (EK1122)/PLC Coupler 2 (EK1100)/PLC Junction 10 (EK1122)/PF1K4-WFS (EK1100)/PF1K4-EL2004-E4
//     PlcTask Outputs/Main.M18.bBrakeRelease <-> Channel 1/Output
//   tmo_motion Instance <-> Device 1 (EtherCAT)/Power (EK1200)/PLC Junction 2 (EK1122)/PLC Coupler 2 (EK1100)/PLC Junction 10 (EK1122)/PF1K4-WFS (EK1100)/PF1K4-EL3314-E5
//     PlcTask Inputs/PRG_PF1K4_WFS_TARGET.fbPF1K4.fbThermoCouple1.bError <-> TC Inputs Channel 1/Status/Error
//     PlcTask Inputs/PRG_PF1K4_WFS_TARGET.fbPF1K4.fbThermoCouple2.bError <-> TC Inputs Channel 2/Status/Error
//     PlcTask Inputs/PRG_PF1K4_WFS_TARGET.fbPF1K4.fbThermoCouple1.bOverrange <-> TC Inputs Channel 1/Status/Overrange
//     PlcTask Inputs/PRG_PF1K4_WFS_TARGET.fbPF1K4.fbThermoCouple2.bOverrange <-> TC Inputs Channel 2/Status/Overrange
//     PlcTask Inputs/PRG_PF1K4_WFS_TARGET.fbPF1K4.fbThermoCouple1.bUnderrange <-> TC Inputs Channel 1/Status/Underrange
//     PlcTask Inputs/PRG_PF1K4_WFS_TARGET.fbPF1K4.fbThermoCouple2.bUnderrange <-> TC Inputs Channel 2/Status/Underrange
//     PlcTask Inputs/PRG_PF1K4_WFS_TARGET.fbPF1K4.fbThermoCouple1.iRaw <-> TC Inputs Channel 1/Value
//     PlcTask Inputs/PRG_PF1K4_WFS_TARGET.fbPF1K4.fbThermoCouple2.iRaw <-> TC Inputs Channel 2/Value
//   tmo_motion Instance <-> Device 1 (EtherCAT)/Power (EK1200)/PLC Junction 2 (EK1122)/PLC Coupler 2 (EK1100)/PLC Junction 10 (EK1122)/PF1K4-WFS (EK1100)/PF1K4-EL5042-E3
//     PlcTask Inputs/Main.M18.nRawEncoderULINT <-> FB Inputs Channel 2/Position
//     PlcTask Inputs/Main.M19.nRawEncoderULINT <-> FB Inputs Channel 1/Position
//   tmo_motion Instance <-> Device 1 (EtherCAT)/Power (EK1200)/PLC Junction 2 (EK1122)/PLC Coupler 2 (EK1100)/PLC Junction 10 (EK1122)/PF1K4-WFS (EK1100)/PF1K4-EL7041-E1
//     PlcTask Inputs/Main.M18.bLimitBackwardEnable <-> STM Status/Status/Digital input 2
//     PlcTask Inputs/Main.M18.bLimitForwardEnable <-> STM Status/Status/Digital input 1
//   tmo_motion Instance <-> Device 1 (EtherCAT)/Power (EK1200)/PLC Junction 2 (EK1122)/PLC Coupler 2 (EK1100)/PLC Junction 7 (EK1122)/TM1K4-ATM (EK1100)/TM1K4-EL2004-E4
//     PlcTask Outputs/Main.M21.bBrakeRelease <-> Channel 1/Output
//   tmo_motion Instance <-> Device 1 (EtherCAT)/Power (EK1200)/PLC Junction 2 (EK1122)/PLC Coupler 2 (EK1100)/PLC Junction 7 (EK1122)/TM1K4-ATM (EK1100)/TM1K4-EL3314-E5
//     PlcTask Inputs/PRG_TM1K4.fbTM1K4.fbThermoCouple1.bError <-> TC Inputs Channel 1/Status/Error
//     PlcTask Inputs/PRG_TM1K4.fbTM1K4.fbThermoCouple1.bOverrange <-> TC Inputs Channel 1/Status/Overrange
//     PlcTask Inputs/PRG_TM1K4.fbTM1K4.fbThermoCouple1.bUnderrange <-> TC Inputs Channel 1/Status/Underrange
//     PlcTask Inputs/PRG_TM1K4.fbTM1K4.fbThermoCouple1.iRaw <-> TC Inputs Channel 1/Value
//   tmo_motion Instance <-> Device 1 (EtherCAT)/Power (EK1200)/PLC Junction 2 (EK1122)/PLC Coupler 2 (EK1100)/PLC Junction 7 (EK1122)/TM1K4-ATM (EK1100)/TM1K4-EL5042-E3
//     PlcTask Inputs/Main.M21.nRawEncoderULINT <-> FB Inputs Channel 1/Position
//     PlcTask Inputs/Main.M22.nRawEncoderULINT <-> FB Inputs Channel 2/Position
//   tmo_motion Instance <-> Device 1 (EtherCAT)/Power (EK1200)/PLC Junction 2 (EK1122)/PLC Coupler 2 (EK1100)/PLC Junction 7 (EK1122)/TM1K4-ATM (EK1100)/TM1K4-EL7041-E1
//     PlcTask Inputs/Main.M21.bLimitBackwardEnable <-> STM Status/Status/Digital input 2
//     PlcTask Inputs/Main.M21.bLimitForwardEnable <-> STM Status/Status/Digital input 1
//   tmo_motion Instance <-> Device 1 (EtherCAT)/Power (EK1200)/PLC Junction 2 (EK1122)/PLC Coupler 2 (EK1100)/PLC Junction 8 (EK1122)/IM5K4-PPM (EK1100)/IM5K4-EL2004-E3
//     PlcTask Outputs/Main.M17.bBrakeRelease <-> Channel 1/Output
//     PlcTask Outputs/PRG_IM5K4_PPM.fbIM5K4.fbGige.bGigePower <-> Channel 2/Output
//   tmo_motion Instance <-> Device 1 (EtherCAT)/Power (EK1200)/PLC Junction 2 (EK1122)/PLC Coupler 2 (EK1100)/PLC Junction 8 (EK1122)/IM5K4-PPM (EK1100)/IM5K4-EL3062-E6
//     PlcTask Inputs/PRG_IM5K4_PPM.fbIM5K4.fbPowerMeter.iVoltageINT <-> AI Standard Channel 1/Value
//   tmo_motion Instance <-> Device 1 (EtherCAT)/Power (EK1200)/PLC Junction 2 (EK1122)/PLC Coupler 2 (EK1100)/PLC Junction 8 (EK1122)/IM5K4-PPM (EK1100)/IM5K4-EL3314-E4
//     PlcTask Inputs/PRG_IM5K4_PPM.fbIM5K4.fbPowerMeter.fbThermoCouple.bError <-> TC Inputs Channel 1/Status/Error
//     PlcTask Inputs/PRG_IM5K4_PPM.fbIM5K4.fbPowerMeter.fbThermoCouple.bOverrange <-> TC Inputs Channel 1/Status/Overrange
//     PlcTask Inputs/PRG_IM5K4_PPM.fbIM5K4.fbPowerMeter.fbThermoCouple.bUnderrange <-> TC Inputs Channel 1/Status/Underrange
//     PlcTask Inputs/PRG_IM5K4_PPM.fbIM5K4.fbPowerMeter.fbThermoCouple.iRaw <-> TC Inputs Channel 1/Value
//     PlcTask Inputs/PRG_IM5K4_PPM.fbIM5K4.fbYagThermoCouple.bError <-> TC Inputs Channel 2/Status/Error
//     PlcTask Inputs/PRG_IM5K4_PPM.fbIM5K4.fbYagThermoCouple.bOverrange <-> TC Inputs Channel 2/Status/Overrange
//     PlcTask Inputs/PRG_IM5K4_PPM.fbIM5K4.fbYagThermoCouple.bUnderrange <-> TC Inputs Channel 2/Status/Underrange
//     PlcTask Inputs/PRG_IM5K4_PPM.fbIM5K4.fbYagThermoCouple.iRaw <-> TC Inputs Channel 2/Value
//   tmo_motion Instance <-> Device 1 (EtherCAT)/Power (EK1200)/PLC Junction 2 (EK1122)/PLC Coupler 2 (EK1100)/PLC Junction 8 (EK1122)/IM5K4-PPM (EK1100)/IM5K4-EL4004-E7
//     PlcTask Outputs/PRG_IM5K4_PPM.fbIM5K4.fbGige.iIlluminatorINT <-> AO Outputs Channel 1/Analog output
//   tmo_motion Instance <-> Device 1 (EtherCAT)/Power (EK1200)/PLC Junction 2 (EK1122)/PLC Coupler 2 (EK1100)/PLC Junction 8 (EK1122)/IM5K4-PPM (EK1100)/IM5K4-EL5042-E2
//     PlcTask Inputs/Main.M17.nRawEncoderULINT <-> FB Inputs Channel 1/Position
//   tmo_motion Instance <-> Device 1 (EtherCAT)/Power (EK1200)/PLC Junction 2 (EK1122)/PLC Coupler 2 (EK1100)/PLC Junction 8 (EK1122)/IM5K4-PPM (EK1100)/IM5K4-EL7041-E1
//     PlcTask Inputs/Main.M17.bLimitBackwardEnable <-> STM Status/Status/Digital input 2
//     PlcTask Inputs/Main.M17.bLimitForwardEnable <-> STM Status/Status/Digital input 1
//   tmo_motion Instance <-> Device 1 (EtherCAT)/Power (EK1200)/PLC Junction 2 (EK1122)/PLC Coupler 2 (EK1100)/PLC Junction 8 (EK1122)/ST4K4-TERM (EP2338-0001)
//     PlcTask Inputs/PRG_ST4K4_TMO_TERM.ST4K4.i_xInsertedLS <-> Channel 4/Input
//     PlcTask Inputs/PRG_ST4K4_TMO_TERM.ST4K4.i_xRetractedLS <-> Channel 3/Input
//     PlcTask Outputs/PRG_ST4K4_TMO_TERM.ST4K4.q_xRetract_DO <-> Channel 9/Output
//   tmo_motion Instance <-> Device 1 (EtherCAT)/Power (EK1200)/PLC Junction 2 (EK1122)/PLC Coupler 2 (EK1100)/PLC Junction 9 (EK1122)/X2 SL2K4-SCATTER/SL2K4-EL5101-E2
//     PlcTask Inputs/Main.M23.nRawEncoderUINT <-> ENC Status compact/Counter value
//   tmo_motion Instance <-> Device 1 (EtherCAT)/Power (EK1200)/PLC Junction 2 (EK1122)/PLC Coupler 2 (EK1100)/PLC Junction 9 (EK1122)/X2 SL2K4-SCATTER/SL2K4-EL5101-E4
//     PlcTask Inputs/Main.M24.nRawEncoderUINT <-> ENC Status compact/Counter value
//   tmo_motion Instance <-> Device 1 (EtherCAT)/Power (EK1200)/PLC Junction 2 (EK1122)/PLC Coupler 2 (EK1100)/PLC Junction 9 (EK1122)/X2 SL2K4-SCATTER/SL2K4-EL5101-E6
//     PlcTask Inputs/Main.M25.nRawEncoderUINT <-> ENC Status compact/Counter value
//   tmo_motion Instance <-> Device 1 (EtherCAT)/Power (EK1200)/PLC Junction 2 (EK1122)/PLC Coupler 2 (EK1100)/PLC Junction 9 (EK1122)/X2 SL2K4-SCATTER/SL2K4-EL5101-E8
//     PlcTask Inputs/Main.M26.nRawEncoderUINT <-> ENC Status compact/Counter value
//   tmo_motion Instance <-> Device 1 (EtherCAT)/Power (EK1200)/PLC Junction 2 (EK1122)/PLC Coupler 2 (EK1100)/PLC Junction 9 (EK1122)/X2 SL2K4-SCATTER/SL2K4-EL7031-E1
//     PlcTask Inputs/Main.M23.bLimitBackwardEnable <-> STM Status/Status/Digital input 1
//     PlcTask Inputs/Main.M23.bLimitForwardEnable <-> STM Status/Status/Digital input 2
//   tmo_motion Instance <-> Device 1 (EtherCAT)/Power (EK1200)/PLC Junction 2 (EK1122)/PLC Coupler 2 (EK1100)/PLC Junction 9 (EK1122)/X2 SL2K4-SCATTER/SL2K4-EL7031-E3
//     PlcTask Inputs/Main.M24.bLimitBackwardEnable <-> STM Status/Status/Digital input 1
//     PlcTask Inputs/Main.M24.bLimitForwardEnable <-> STM Status/Status/Digital input 2
//   tmo_motion Instance <-> Device 1 (EtherCAT)/Power (EK1200)/PLC Junction 2 (EK1122)/PLC Coupler 2 (EK1100)/PLC Junction 9 (EK1122)/X2 SL2K4-SCATTER/SL2K4-EL7031-E5
//     PlcTask Inputs/Main.M25.bLimitBackwardEnable <-> STM Status/Status/Digital input 2
//     PlcTask Inputs/Main.M25.bLimitForwardEnable <-> STM Status/Status/Digital input 1
//   tmo_motion Instance <-> Device 1 (EtherCAT)/Power (EK1200)/PLC Junction 2 (EK1122)/PLC Coupler 2 (EK1100)/PLC Junction 9 (EK1122)/X2 SL2K4-SCATTER/SL2K4-EL7031-E7
//     PlcTask Inputs/Main.M26.bLimitBackwardEnable <-> STM Status/Status/Digital input 2
//     PlcTask Inputs/Main.M26.bLimitForwardEnable <-> STM Status/Status/Digital input 1
//   tmo_motion Instance <-> Device 1 (EtherCAT)/Power (EK1200)/PMPS_FFO
//     PlcTask Outputs/GVL_PMPS.fbFastFaultOutput1.q_xFastFaultOut <-> Channel 1/Output
//     PlcTask Outputs/GVL_PMPS.fbFastFaultOutput2.q_xFastFaultOut <-> Channel 2/Output
//   tmo_motion Instance <-> Device 1 (EtherCAT)/Power (EK1200)/PMPS_PRE
//     PlcTask Inputs/PRG_3_PMPS_POST.fbArbiterIO.i_stCurrentBP <-> IO Inputs/CurrentBP
//     PlcTask Inputs/PRG_3_PMPS_POST.fbArbiterIO.xTxPDO_state <-> SYNC Inputs/TxPDO state
//     PlcTask Inputs/PRG_3_PMPS_POST.fbArbiterIO.xTxPDO_toggle <-> SYNC Inputs/TxPDO toggle
//     PlcTask Outputs/PRG_3_PMPS_POST.fbArbiterIO.q_stRequestedBP <-> IO Outputs/RequestedBP
//   tmo_motion Instance <-> NC-Task 1 SAF/Axes/Axis 1 AL1K4-L2SI-MMS
//     PlcTask Inputs/Main.M1.Axis.NcToPlc <-> Outputs/ToPlc
//     PlcTask Outputs/Main.M1.Axis.PlcToNc <-> Inputs/FromPlc
//   tmo_motion Instance <-> NC-Task 1 SAF/Axes/Axis 15 IM3K4-PPM-MMS
//     PlcTask Inputs/Main.M15.Axis.NcToPlc <-> Outputs/ToPlc
//     PlcTask Outputs/Main.M15.Axis.PlcToNc <-> Inputs/FromPlc
//   tmo_motion Instance <-> NC-Task 1 SAF/Axes/Axis 16 IM4K4-PPM-MMS
//     PlcTask Inputs/Main.M16.Axis.NcToPlc <-> Outputs/ToPlc
//     PlcTask Outputs/Main.M16.Axis.PlcToNc <-> Inputs/FromPlc
//   tmo_motion Instance <-> NC-Task 1 SAF/Axes/Axis 17 IM5K4-PPM-MMS
//     PlcTask Inputs/Main.M17.Axis.NcToPlc <-> Outputs/ToPlc
//     PlcTask Outputs/Main.M17.Axis.PlcToNc <-> Inputs/FromPlc
//   tmo_motion Instance <-> NC-Task 1 SAF/Axes/Axis 18 PF1K4-WFS_TARGET-MMS-Y
//     PlcTask Inputs/Main.M18.Axis.NcToPlc <-> Outputs/ToPlc
//     PlcTask Outputs/Main.M18.Axis.PlcToNc <-> Inputs/FromPlc
//   tmo_motion Instance <-> NC-Task 1 SAF/Axes/Axis 19 PF1K4-WFS_TARGET-MMS-Z
//     PlcTask Inputs/Main.M19.Axis.NcToPlc <-> Outputs/ToPlc
//     PlcTask Outputs/Main.M19.Axis.PlcToNc <-> Inputs/FromPlc
//   tmo_motion Instance <-> NC-Task 1 SAF/Axes/Axis 2
//     PlcTask Inputs/Main.M2.Axis.NcToPlc <-> Outputs/ToPlc
//     PlcTask Outputs/Main.M2.Axis.PlcToNc <-> Inputs/FromPlc
//   tmo_motion Instance <-> NC-Task 1 SAF/Axes/Axis 20 LI1K4-IP1-MMS
//     PlcTask Inputs/Main.M20.Axis.NcToPlc <-> Outputs/ToPlc
//     PlcTask Outputs/Main.M20.Axis.PlcToNc <-> Inputs/FromPlc
//   tmo_motion Instance <-> NC-Task 1 SAF/Axes/Axis 21 TM1K4-MMS-Y
//     PlcTask Inputs/Main.M21.Axis.NcToPlc <-> Outputs/ToPlc
//     PlcTask Outputs/Main.M21.Axis.PlcToNc <-> Inputs/FromPlc
//   tmo_motion Instance <-> NC-Task 1 SAF/Axes/Axis 22 TM1K4-MMS-X
//     PlcTask Inputs/Main.M22.Axis.NcToPlc <-> Outputs/ToPlc
//     PlcTask Outputs/Main.M22.Axis.PlcToNc <-> Inputs/FromPlc
//   tmo_motion Instance <-> NC-Task 1 SAF/Axes/Axis 3
//     PlcTask Inputs/Main.M3.Axis.NcToPlc <-> Outputs/ToPlc
//     PlcTask Outputs/Main.M3.Axis.PlcToNc <-> Inputs/FromPlc
//   tmo_motion Instance <-> NC-Task 1 SAF/Axes/Axis 4
//     PlcTask Inputs/Main.M4.Axis.NcToPlc <-> Outputs/ToPlc
//     PlcTask Outputs/Main.M4.Axis.PlcToNc <-> Inputs/FromPlc
//   tmo_motion Instance <-> NC-Task 1 SAF/Axes/Axis 5
//     PlcTask Inputs/Main.M5.Axis.NcToPlc <-> Outputs/ToPlc
//     PlcTask Outputs/Main.M5.Axis.PlcToNc <-> Inputs/FromPlc
//   tmo_motion Instance <-> NC-Task 1 SAF/Axes/Axis 6 IM1K4-XTES-MMS
//     PlcTask Inputs/Main.M6.Axis.NcToPlc <-> Outputs/ToPlc
//     PlcTask Outputs/Main.M6.Axis.PlcToNc <-> Inputs/FromPlc
//   tmo_motion Instance <-> NC-Task 1 SAF/Axes/Axis 7 IM1K4-XTES-CLZ
//     PlcTask Inputs/Main.M7.Axis.NcToPlc <-> Outputs/ToPlc
//     PlcTask Outputs/Main.M7.Axis.PlcToNc <-> Inputs/FromPlc
//   tmo_motion Instance <-> NC-Task 1 SAF/Axes/Axis 8 IM1K4-XTES-CLF
//     PlcTask Inputs/Main.M8.Axis.NcToPlc <-> Outputs/ToPlc
//     PlcTask Outputs/Main.M8.Axis.PlcToNc <-> Inputs/FromPlc
//   tmo_motion Instance <-> NC-Task 1 SAF/Axes/Axis 9 IM2K4-PPM-MMS
//     PlcTask Inputs/Main.M9.Axis.NcToPlc <-> Outputs/ToPlc
//     PlcTask Outputs/Main.M9.Axis.PlcToNc <-> Inputs/FromPlc
//   tmo_motion Instance <-> NC-Task 1 SAF/Axes/SL1K4-BOTTOM-M10
//     PlcTask Inputs/Main.M10.Axis.NcToPlc <-> Outputs/ToPlc
//     PlcTask Outputs/Main.M10.Axis.PlcToNc <-> Inputs/FromPlc
//   tmo_motion Instance <-> NC-Task 1 SAF/Axes/SL1K4-NORTH-M12
//     PlcTask Inputs/Main.M12.Axis.NcToPlc <-> Outputs/ToPlc
//     PlcTask Outputs/Main.M12.Axis.PlcToNc <-> Inputs/FromPlc
//   tmo_motion Instance <-> NC-Task 1 SAF/Axes/SL1K4-SOUTH-M13
//     PlcTask Inputs/Main.M13.Axis.NcToPlc <-> Outputs/ToPlc
//     PlcTask Outputs/Main.M13.Axis.PlcToNc <-> Inputs/FromPlc
//   tmo_motion Instance <-> NC-Task 1 SAF/Axes/SL1K4-TOP-M11
//     PlcTask Inputs/Main.M11.Axis.NcToPlc <-> Outputs/ToPlc
//     PlcTask Outputs/Main.M11.Axis.PlcToNc <-> Inputs/FromPlc
//   tmo_motion Instance <-> NC-Task 1 SAF/Axes/SL2K4-BOTTOM-M23
//     PlcTask Inputs/Main.M23.Axis.NcToPlc <-> Outputs/ToPlc
//     PlcTask Outputs/Main.M23.Axis.PlcToNc <-> Inputs/FromPlc
//   tmo_motion Instance <-> NC-Task 1 SAF/Axes/SL2K4-NORTH-M25
//     PlcTask Inputs/Main.M25.Axis.NcToPlc <-> Outputs/ToPlc
//     PlcTask Outputs/Main.M25.Axis.PlcToNc <-> Inputs/FromPlc
//   tmo_motion Instance <-> NC-Task 1 SAF/Axes/SL2K4-SOUTH-M26
//     PlcTask Inputs/Main.M26.Axis.NcToPlc <-> Outputs/ToPlc
//     PlcTask Outputs/Main.M26.Axis.PlcToNc <-> Inputs/FromPlc
//   tmo_motion Instance <-> NC-Task 1 SAF/Axes/SL2K4-TOP-M24
//     PlcTask Inputs/Main.M24.Axis.NcToPlc <-> Outputs/ToPlc
//     PlcTask Outputs/Main.M24.Axis.PlcToNc <-> Inputs/FromPlc
//   tmo_motion Instance <-> NC-Task 1 SAF/Axes/ST1K4-TEST
//     PlcTask Inputs/Main.M14.Axis.NcToPlc <-> Outputs/ToPlc
//     PlcTask Outputs/Main.M14.Axis.PlcToNc <-> Inputs/FromPlc

CONFIGURATION tmo_motion
    RESOURCE PLC ON TwinCAT3
        TASK PlcTask(INTERVAL := T#10ms, PRIORITY := 20);
        PROGRAM PRG_1_PlcTask WITH PlcTask : PRG_1_PlcTask;
    END_RESOURCE
END_CONFIGURATION

// ---- GVLs/Main.TcGVL
{attribute 'qualified_only'}
VAR_GLOBAL
    // AL1K4-L2SI: 1 Axis
    {attribute 'pytmc' := 'pv: AL1K4:L2SI:MMS'}
    {attribute 'TcLinkTo' := '.bLimitForwardEnable  := TIIB[AL1K4-EL7041-E1]^STM Status^Status^Digital input 1;
                              .bLimitBackwardEnable := TIIB[AL1K4-EL7041-E1]^STM Status^Status^Digital input 2;
                              .bBrakeRelease        := TIIB[AL1K4-EL2004-E3]^Channel 1^Output;
                              .nRawEncoderULINT     := TIIB[AL1K4-EL5042-E2]^FB Inputs Channel 1^Position'}
    M1: DUT_MotionStage := (sName := 'AL1K4:L2SI:MMS');

    // SPARE: 7 Axes (formerly AT1K4-SOLID and IM1K4-XTES)
    M2: DUT_MotionStage;
    M3: DUT_MotionStage;
    M4: DUT_MotionStage;
    M5: DUT_MotionStage;
    M6: DUT_MotionStage;
    M7: DUT_MotionStage;
    M8: DUT_MotionStage;

    // IM2K4-PPM: 1 Axis
    {attribute 'pytmc' := 'pv: IM2K4:PPM:MMS'}
    {attribute 'TcLinkTo' := '.bLimitForwardEnable  := TIIB[IM2K4-EL7041-E1]^STM Status^Status^Digital input 1;
                              .bLimitBackwardEnable := TIIB[IM2K4-EL7041-E1]^STM Status^Status^Digital input 2;
                              .bBrakeRelease        := TIIB[IM2K4-EL2004-E3]^Channel 1^Output;
                              .nRawEncoderULINT     := TIIB[IM2K4-EL5042-E2]^FB Inputs Channel 1^Position'}
    M9: DUT_MotionStage := (sName := 'IM2K4:PPM:MMS');

    // SL1K4-SCATTER: 4 Axes
    {attribute 'pytmc' := 'pv: SL1K4:SCATTER:MMS:BOTTOM'}
    {attribute 'TcLinkTo' := '.bLimitForwardEnable  := TIIB[SL1K4-EL7031-E1]^STM Status^Status^Digital input 2;
                              .bLimitBackwardEnable := TIIB[SL1K4-EL7031-E1]^STM Status^Status^Digital input 1;
                              .nRawEncoderUINT      := TIIB[SL1K4-EL5101-E2]^ENC Status compact^Counter value'}
    M10: DUT_MotionStage := (sName := 'SL1K4:SCATTER:MMS:BOTTOM');
    {attribute 'pytmc' := 'pv: SL1K4:SCATTER:MMS:TOP'}
    {attribute 'TcLinkTo' := '.bLimitForwardEnable  := TIIB[SL1K4-EL7031-E3]^STM Status^Status^Digital input 2;
                              .bLimitBackwardEnable := TIIB[SL1K4-EL7031-E3]^STM Status^Status^Digital input 1;
                              .nRawEncoderUINT      := TIIB[SL1K4-EL5101-E4]^ENC Status compact^Counter value'}
    M11: DUT_MotionStage := (sName := 'SL1K4:SCATTER:MMS:TOP');
    {attribute 'pytmc' := 'pv: SL1K4:SCATTER:MMS:NORTH'}
    {attribute 'TcLinkTo' := '.bLimitForwardEnable  := TIIB[SL1K4-EL7031-E5]^STM Status^Status^Digital input 1;
                              .bLimitBackwardEnable := TIIB[SL1K4-EL7031-E5]^STM Status^Status^Digital input 2;
                              .nRawEncoderUINT      := TIIB[SL1K4-EL5101-E6]^ENC Status compact^Counter value'}
    M12: DUT_MotionStage := (sName := 'SL1K4:SCATTER:MMS:NORTH');
    {attribute 'pytmc' := 'pv: SL1K4:SCATTER:MMS:SOUTH'}
    {attribute 'TcLinkTo' := '.bLimitForwardEnable  := TIIB[SL1K4-EL7031-E7]^STM Status^Status^Digital input 1;
                              .bLimitBackwardEnable := TIIB[SL1K4-EL7031-E7]^STM Status^Status^Digital input 2;
                              .nRawEncoderUINT      := TIIB[SL1K4-EL5101-E8]^ENC Status compact^Counter value'}
    M13: DUT_MotionStage := (sName := 'SL1K4:SCATTER:MMS:SOUTH');

    // SPARE: 1 Axis (formerly ST1K4-TEST)
    M14: DUT_MotionStage;

    // IM3K4-PPM: 1 Axis
    {attribute 'pytmc' := 'pv: IM3K4:PPM:MMS'}
    {attribute 'TcLinkTo' := '.bLimitForwardEnable  := TIIB[IM3K4-EL7041-E1]^STM Status^Status^Digital input 1;
                              .bLimitBackwardEnable := TIIB[IM3K4-EL7041-E1]^STM Status^Status^Digital input 2;
                              .bBrakeRelease        := TIIB[IM3K4-EL2004-E3]^Channel 1^Output;
                              .nRawEncoderULINT     := TIIB[IM3K4-EL5042-E2]^FB Inputs Channel 1^Position'}
    M15: DUT_MotionStage := (sName := 'IM3K4:PPM:MMS');
    // IM4K4-PPM: 1 Axis
    {attribute 'pytmc' := 'pv: IM4K4:PPM:MMS'}
    {attribute 'TcLinkTo' := '.bLimitForwardEnable  := TIIB[IM4K4-EL7041-E1]^STM Status^Status^Digital input 1;
                              .bLimitBackwardEnable := TIIB[IM4K4-EL7041-E1]^STM Status^Status^Digital input 2;
                              .bBrakeRelease        := TIIB[IM4K4-EL2004-E3]^Channel 1^Output;
                              .nRawEncoderULINT     := TIIB[IM4K4-EL5042-E2]^FB Inputs Channel 1^Position'}
    M16: DUT_MotionStage := (sName := 'IM4K4:PPM:MMS');

    // IM5K4-PPM: 1 Axis
    {attribute 'pytmc' := 'pv: IM5K4:PPM:MMS'}
    {attribute 'TcLinkTo' := '.bLimitForwardEnable  := TIIB[IM5K4-EL7041-E1]^STM Status^Status^Digital input 1;
                              .bLimitBackwardEnable := TIIB[IM5K4-EL7041-E1]^STM Status^Status^Digital input 2;
                              .bBrakeRelease        := TIIB[IM5K4-EL2004-E3]^Channel 1^Output;
                              .nRawEncoderULINT     := TIIB[IM5K4-EL5042-E2]^FB Inputs Channel 1^Position'}
    M17: DUT_MotionStage := (sName := 'IM5K4:PPM:MMS');

    // PF1K4-WFS_TARGET: 2 Axes
    {attribute 'pytmc' := 'pv: PF1K4:WFS:MMS:Y'}
    {attribute 'TcLinkTo' := '.bLimitForwardEnable  := TIIB[PF1K4-EL7041-E1]^STM Status^Status^Digital input 1;
                              .bLimitBackwardEnable := TIIB[PF1K4-EL7041-E1]^STM Status^Status^Digital input 2;
                              .bBrakeRelease        := TIIB[PF1K4-EL2004-E4]^Channel 1^Output;
                              .nRawEncoderULINT     := TIIB[PF1K4-EL5042-E3]^FB Inputs Channel 2^Position'}
    M18: DUT_MotionStage := (sName := 'PF1K4:WFS:MMS:Y');
    {attribute 'pytmc' := 'pv: PF1K4:WFS:MMS:Z'}
    {attribute 'TcLinkTo' := '.nRawEncoderULINT     := TIIB[PF1K4-EL5042-E3]^FB Inputs Channel 1^Position'}
    M19: DUT_MotionStage := (sName := 'PF1K4:WFS:MMS:Z');

    // LI1K4-IP1: 1 Axis
    {attribute 'pytmc' := 'pv: LI1K4:IP1:MMS'}
    {attribute 'TcLinkTo' := '.bLimitForwardEnable  := TIIB[LI1K4-EL7041-E1]^STM Status^Status^Digital input 1;
                              .bLimitBackwardEnable := TIIB[LI1K4-EL7041-E1]^STM Status^Status^Digital input 2;
                              .bBrakeRelease        := TIIB[LI1K4-EL2004-E3]^Channel 1^Output;
                              .nRawEncoderULINT     := TIIB[LI1K4-EL5042-E2]^FB Inputs Channel 1^Position'}
    M20: DUT_MotionStage := (sName := 'LI1K4:IP1:MMS');

    // TM1K4: 2 Axes
    {attribute 'pytmc' := 'pv: TM1K4:ATM:MMS:Y'}
    {attribute 'TcLinkTo' := '.bLimitForwardEnable  := TIIB[TM1K4-EL7041-E1]^STM Status^Status^Digital input 1;
                              .bLimitBackwardEnable := TIIB[TM1K4-EL7041-E1]^STM Status^Status^Digital input 2;
                              .bBrakeRelease        := TIIB[TM1K4-EL2004-E4]^Channel 1^Output;
                              .nRawEncoderULINT     := TIIB[TM1K4-EL5042-E3]^FB Inputs Channel 1^Position'}
    M21: DUT_MotionStage := (sName := 'TM1K4:ATM:MMS:Y');
    {attribute 'pytmc' := 'pv: TM1K4:ATM:MMS:X'}
    {attribute 'TcLinkTo' := '.nRawEncoderULINT     := TIIB[TM1K4-EL5042-E3]^FB Inputs Channel 2^Position'}
    M22: DUT_MotionStage := (sName := 'TM1K4:ATM:MMS:X');

     // SL2K4-SCATTER: 4 Axes
    {attribute 'pytmc' := 'pv: SL2K4:SCATTER:MMS:BOTTOM'}
    {attribute 'TcLinkTo' := '.bLimitForwardEnable  := TIIB[SL2K4-EL7031-E1]^STM Status^Status^Digital input 2;
                             .bLimitBackwardEnable := TIIB[SL2K4-EL7031-E1]^STM Status^Status^Digital input 1;
                              .nRawEncoderUINT      := TIIB[SL2K4-EL5101-E2]^ENC Status compact^Counter value'}
    M23: DUT_MotionStage := (sName := 'SL2K4:SCATTER:MMS:BOTTOM');
    {attribute 'pytmc' := 'pv: SL2K4:SCATTER:MMS:TOP'}
    {attribute 'TcLinkTo' := '.bLimitForwardEnable  := TIIB[SL2K4-EL7031-E3]^STM Status^Status^Digital input 2;
                              .bLimitBackwardEnable := TIIB[SL2K4-EL7031-E3]^STM Status^Status^Digital input 1;
                              .nRawEncoderUINT      := TIIB[SL2K4-EL5101-E4]^ENC Status compact^Counter value'}
    M24: DUT_MotionStage := (sName := 'SL2K4:SCATTER:MMS:TOP');
    {attribute 'pytmc' := 'pv: SL2K4:SCATTER:MMS:NORTH'}
    {attribute 'TcLinkTo' := '.bLimitForwardEnable  := TIIB[SL2K4-EL7031-E5]^STM Status^Status^Digital input 1;
                              .bLimitBackwardEnable := TIIB[SL2K4-EL7031-E5]^STM Status^Status^Digital input 2;
                              .nRawEncoderUINT      := TIIB[SL2K4-EL5101-E6]^ENC Status compact^Counter value'}
    M25: DUT_MotionStage := (sName := 'SL2K4:SCATTER:MMS:NORTH');
    {attribute 'pytmc' := 'pv: SL2K4:SCATTER:MMS:SOUTH'}
    {attribute 'TcLinkTo' := '.bLimitForwardEnable  := TIIB[SL2K4-EL7031-E7]^STM Status^Status^Digital input 1;
                              .bLimitBackwardEnable := TIIB[SL2K4-EL7031-E7]^STM Status^Status^Digital input 2;
                              .nRawEncoderUINT      := TIIB[SL2K4-EL5101-E8]^ENC Status compact^Counter value'}
    M26: DUT_MotionStage := (sName := 'SL2K4:SCATTER:MMS:SOUTH');
END_VAR

// ---- POUs/PRG_1_PlcTask.TcPOU
PROGRAM PRG_1_PlcTask
VAR
END_VAR

PRG_2_PMPS_PRE();

PRG_AL1K4_L2SI();
PRG_IM2K4_PPM();
PRG_IM3K4_PPM();
PRG_IM4K4_PPM();
PRG_IM5K4_PPM();
PRG_LI1K4_IP1();
PRG_PF1K4_WFS_TARGET();
PRG_SL1K4_SCATTER();
PRG_SL2K4_SCATTER();
PRG_ST4K4_TMO_TERM();
PRG_ST5K4_TMO_TERM_FIXED();
PRG_TM1K4();

PRG_3_PMPS_POST();
PRG_4_LOG();

END_PROGRAM

// ---- POUs/PRG_2_PMPS_PRE.TcPOU
PROGRAM PRG_2_PMPS_PRE
VAR
END_VAR

END_PROGRAM

// ---- POUs/PRG_AL1K4_L2SI.TcPOU
PROGRAM PRG_AL1K4_L2SI
VAR
    {attribute 'pytmc' := '
        pv: AL1K4:L2SI
        io: io
    '}
    {attribute 'TcLinkTo' := '.fbLaser.iLaserINT := TIIB[AL1K4-EL4004-E4]^AO Outputs Channel 1^Analog output;
                              .fbLaser.iShutdownINT := TIIB[AL1K4-EL4004-E4]^AO Outputs Channel 2^Analog output'}
    fbAL1K4: FB_REF;
END_VAR

fbAL1K4.nTransitionAssertionID := 16#6140;
fbAL1K4.nUnknownAssertionID := 16#6149;

